// ---- Visualizations/Visualizations/Maintenance_2.TcVIS
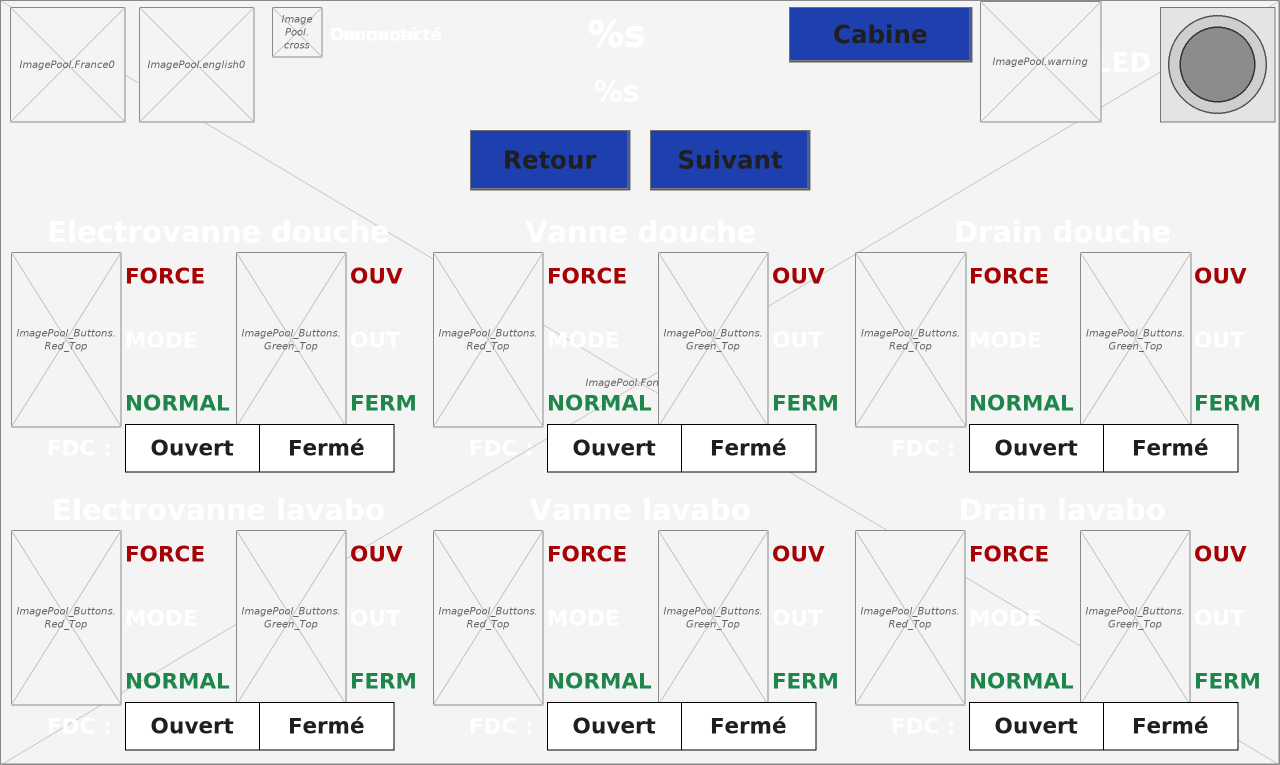
VISUALIZATION Maintenance_2  // 1280x765
    Frame (0,0 1280x765)
        shows masque()
    Button (650,130 160x60), "Suivant"
        OnMouseDown: execute {
            IF (Option_Bas_Debit OR Option_Douchette OR Option_NEP)
            	THEN
            	VisuElems.CURRENTVISU := 'Maintenance_3';
            	ELSIF (Option_WC_GV OR Option_WC_PV OR Option_Prise)
            		THEN
            		VisuElems.CURRENTVISU := 'Maintenance_4';
            	ELSIF (Option_Cabine_Climatique)
            		THEN
            		VisuElems.CURRENTVISU := 'Maintenance_5';
            	ELSIF (Option_Com_RegSouf_Ultrason)
            		THEN
            		VisuElems.CURRENTVISU := 'Maintenance_6';
            	ELSE
            		VisuElems.CURRENTVISU := 'Maintenance_7';
            END_IF
        }
    Button (470,130 160x60), "Retour"
        OnMouseDown: execute {
            IF (Option_RegSouf_Ultrason OR Option_Reg_Etanche_Ext OR Option_V3V_EauMitig)
            	THEN
            	VisuElems.CURRENTVISU := 'Maintenance_1';
            	ELSE
            	VisuElems.CURRENTVISU := 'menu';
            END_IF
        }
    Group (433,212 415x260), invisible if: NOT Option_Douche OR Option_Debitmetre_Douche
        Group (0,40 415x174)
            Group (0,0 225x175)
                Group (0,0 110x175)
                    Image (0,0 110x175), invisible if: EF_Cmd_Vanne_Alim_Douche, image: ImagePool_Buttons.Green_Bottom
                        OnMouseDown: toggle EF_Cmd_Vanne_Alim_Douche
                    Image (0,0 110x175), invisible if: NOT EF_Cmd_Vanne_Alim_Douche, image: ImagePool_Buttons.Red_Top
                        OnMouseDown: toggle EF_Cmd_Vanne_Alim_Douche
                Rectangle (111,0 114x48), "FORCE"
                Rectangle (111,64 114x48), "MODE"
                Rectangle (111,127 114x48), "NORMAL"
            Group (225,0 190x175), invisible if: NOT EF_Cmd_Vanne_Alim_Douche
                Group (0,0 110x175)
                    Image (0,0 110x175), invisible if: F_Cmd_Vanne_Alim_Douche, image: ImagePool_Buttons.Red_Bottom
                        OnMouseDown: toggle F_Cmd_Vanne_Alim_Douche
                    Image (0,0 110x175), invisible if: NOT F_Cmd_Vanne_Alim_Douche, image: ImagePool_Buttons.Green_Top
                        OnMouseDown: toggle F_Cmd_Vanne_Alim_Douche
                Rectangle (111,0 79x48), "OUV"
                Rectangle (111,64 79x48), "OUT"
                Rectangle (111,127 79x48), "FERM"
        Group (33,212 350x48)
            Rectangle (0,0 81x48), "FDC :"
            RoundedRectangle (81,0 135x48), "Ouvert", invisible if: NOT E_Vanne_Alim_Douche_Ouv
            RoundedRectangle (215,0 135x48), "Fermé", invisible if: NOT E_Vanne_Alim_Douche_Ferm
        Rectangle (0,0 415x40), "Vanne douche"
    Group (433,490 415x260), invisible if: NOT Option_Lavabo OR Option_Debitmetre_Lavabo
        Group (0,40 415x174)
            Group (0,0 225x175)
                Group (0,0 110x175)
                    Image (0,0 110x175), invisible if: EF_Cmd_Vanne_Alim_Douche, image: ImagePool_Buttons.Green_Bottom
                        OnMouseDown: toggle EF_Cmd_Vanne_Alim_Douche
                    Image (0,0 110x175), invisible if: NOT EF_Cmd_Vanne_Alim_Douche, image: ImagePool_Buttons.Red_Top
                        OnMouseDown: toggle EF_Cmd_Vanne_Alim_Douche
                Rectangle (111,0 114x48), "FORCE"
                Rectangle (111,64 114x48), "MODE"
                Rectangle (111,127 114x48), "NORMAL"
            Group (225,0 190x175), invisible if: NOT EF_Cmd_Vanne_Alim_Douche
                Group (0,0 110x175)
                    Image (0,0 110x175), invisible if: F_Cmd_Vanne_Alim_Douche, image: ImagePool_Buttons.Red_Bottom
                        OnMouseDown: toggle F_Cmd_Vanne_Alim_Douche
                    Image (0,0 110x175), invisible if: NOT F_Cmd_Vanne_Alim_Douche, image: ImagePool_Buttons.Green_Top
                        OnMouseDown: toggle F_Cmd_Vanne_Alim_Douche
                Rectangle (111,0 79x48), "OUV"
                Rectangle (111,64 79x48), "OUT"
                Rectangle (111,127 79x48), "FERM"
        Group (33,212 350x48)
            Rectangle (0,0 81x48), "FDC :"
            RoundedRectangle (81,0 135x48), "Ouvert", invisible if: NOT E_Vanne_Alim_Lavabo_Ouv
            RoundedRectangle (215,0 135x48), "Fermé", invisible if: NOT E_Vanne_Alim_Lavabo_Ferm
        Rectangle (0,0 415x40), "Vanne lavabo"
    Group (855,212 415x260), invisible if: NOT Option_Douche
        Group (0,40 415x174)
            Group (0,0 225x175)
                Group (0,0 110x175)
                    Image (0,0 111x175), invisible if: EF_Cmd_Vanne_Vid_Douche, image: ImagePool_Buttons.Green_Bottom
                        OnMouseDown: toggle EF_Cmd_Vanne_Vid_Douche
                    Image (0,0 111x175), invisible if: NOT EF_Cmd_Vanne_Vid_Douche, image: ImagePool_Buttons.Red_Top
                        OnMouseDown: toggle EF_Cmd_Vanne_Vid_Douche
                Rectangle (111,0 114x48), "FORCE"
                Rectangle (111,64 114x48), "MODE"
                Rectangle (111,127 114x48), "NORMAL"
            Group (225,0 190x175), invisible if: NOT EF_Cmd_Vanne_Vid_Douche
                Group (0,0 110x175)
                    Image (0,0 111x175), invisible if: F_Cmd_Vanne_Vid_Douche, image: ImagePool_Buttons.Red_Bottom
                        OnMouseDown: toggle F_Cmd_Vanne_Vid_Douche
                    Image (0,0 111x175), invisible if: NOT F_Cmd_Vanne_Vid_Douche, image: ImagePool_Buttons.Green_Top
                        OnMouseDown: toggle F_Cmd_Vanne_Vid_Douche
                Rectangle (111,0 79x48), "OUV"
                Rectangle (111,64 79x48), "OUT"
                Rectangle (111,127 79x48), "FERM"
        Group (33,212 350x48)
            Rectangle (0,0 81x48), "FDC :"
            RoundedRectangle (81,0 135x48), "Ouvert", invisible if: NOT E_Vanne_Vidange_Douche_Ouv
            RoundedRectangle (215,0 135x48), "Fermé", invisible if: NOT E_Vanne_Vidange_Douche_Ferm
        Rectangle (0,0 415x40), "Drain douche"
    Group (855,490 415x260), invisible if: NOT Option_Lavabo
        Group (0,40 415x174)
            Group (0,0 225x175)
                Group (0,0 110x175)
                    Image (0,0 110x175), invisible if: EF_Cmd_Vanne_Vid_Lavabo, image: ImagePool_Buttons.Green_Bottom
                        OnMouseDown: toggle EF_Cmd_Vanne_Vid_Lavabo
                    Image (0,0 110x175), invisible if: NOT EF_Cmd_Vanne_Vid_Lavabo, image: ImagePool_Buttons.Red_Top
                        OnMouseDown: toggle EF_Cmd_Vanne_Vid_Lavabo
                Rectangle (111,0 114x48), "FORCE"
                Rectangle (111,64 114x48), "MODE"
                Rectangle (111,127 114x48), "NORMAL"
            Group (225,0 190x175), invisible if: NOT EF_Cmd_Vanne_Vid_Lavabo
                Group (0,0 110x175)
                    Image (0,0 110x175), invisible if: F_Cmd_Vanne_Vid_Lavabo, image: ImagePool_Buttons.Red_Bottom
                        OnMouseDown: toggle F_Cmd_Vanne_Vid_Lavabo
                    Image (0,0 110x175), invisible if: NOT F_Cmd_Vanne_Vid_Lavabo, image: ImagePool_Buttons.Green_Top
                        OnMouseDown: toggle F_Cmd_Vanne_Vid_Lavabo
                Rectangle (111,0 79x48), "OUV"
                Rectangle (111,64 79x48), "OUT"
                Rectangle (111,127 79x48), "FERM"
        Group (33,212 350x48)
            Rectangle (0,0 81x48), "FDC :"
            RoundedRectangle (81,0 135x48), "Ouvert", invisible if: NOT E_Vanne_Vidange_Lavabo_Ouv
            RoundedRectangle (215,0 135x48), "Fermé", invisible if: NOT E_Vanne_Vidange_Lavabo_Ferm
        Rectangle (0,0 415x40), "Drain lavabo"
    Group (11,212 415x260), invisible if: NOT Option_Douche OR NOT Option_Debitmetre_Douche
        Group (0,40 415x174)
            Group (0,0 225x175)
                Group (0,0 110x175)
                    Image (0,0 110x175), invisible if: EF_Cmd_ElectroValve_Alim_Douche, image: ImagePool_Buttons.Green_Bottom
                    Image (0,0 110x175), invisible if: NOT EF_Cmd_ElectroValve_Alim_Douche, image: ImagePool_Buttons.Red_Top
                Rectangle (111,0 114x48), "FORCE"
                Rectangle (111,64 114x48), "MODE"
                Rectangle (111,127 114x48), "NORMAL"
            Group (225,0 190x175), invisible if: NOT EF_Cmd_ElectroValve_Alim_Douche
                Group (0,0 110x175)
                    Image (0,0 110x175), invisible if: F_Cmd_ElectroValve_Alim_Douche, image: ImagePool_Buttons.Red_Bottom
                        OnMouseDown: toggle F_Cmd_ElectroValve_Alim_Douche
                    Image (0,0 110x175), invisible if: NOT F_Cmd_ElectroValve_Alim_Douche, image: ImagePool_Buttons.Green_Top
                        OnMouseDown: toggle F_Cmd_ElectroValve_Alim_Douche
                Rectangle (111,0 79x48), "OUV"
                Rectangle (111,64 79x48), "OUT"
                Rectangle (111,127 79x48), "FERM"
        Group (33,212 350x48), invisible if: TRUE
            Rectangle (0,0 81x48), "FDC :"
            RoundedRectangle (81,0 135x48), "Ouvert"
            RoundedRectangle (215,0 135x48), "Fermé"
        Rectangle (0,0 415x40), "Electrovanne douche"
    Group (11,490 415x260), invisible if: NOT Option_Lavabo OR NOT Option_Debitmetre_Lavabo
        Group (0,40 415x174)
            Group (0,0 225x175)
                Group (0,0 110x175)
                    Image (0,0 110x175), invisible if: EF_Cmd_ElectroValve_Alim_Lavabo, image: ImagePool_Buttons.Green_Bottom
                        OnMouseDown: toggle EF_Cmd_ElectroValve_Alim_Lavabo
                    Image (0,0 110x175), invisible if: NOT EF_Cmd_ElectroValve_Alim_Lavabo, image: ImagePool_Buttons.Red_Top
                        OnMouseDown: toggle EF_Cmd_ElectroValve_Alim_Lavabo
                Rectangle (111,0 114x48), "FORCE"
                Rectangle (111,64 114x48), "MODE"
                Rectangle (111,127 114x48), "NORMAL"
            Group (225,0 190x175), invisible if: NOT EF_Cmd_ElectroValve_Alim_Lavabo
                Group (0,0 110x175)
                    Image (0,0 110x175), invisible if: F_Cmd_ElectroValve_Alim_Lavabo, image: ImagePool_Buttons.Red_Bottom
                        OnMouseDown: toggle F_Cmd_ElectroValve_Alim_Lavabo
                    Image (0,0 110x175), invisible if: NOT F_Cmd_ElectroValve_Alim_Lavabo, image: ImagePool_Buttons.Green_Top
                        OnMouseDown: toggle F_Cmd_ElectroValve_Alim_Lavabo
                Rectangle (111,0 79x48), "OUV"
                Rectangle (111,64 79x48), "OUT"
                Rectangle (111,127 79x48), "FERM"
        Group (33,212 350x48), invisible if: TRUE
            Rectangle (0,0 81x48), "FDC :"
            RoundedRectangle (81,0 135x48), "Ouvert"
            RoundedRectangle (215,0 135x48), "Fermé"
        Rectangle (0,0 415x40), "Electrovanne lavabo"
END_VISUALIZATION

// ---- Visualizations/Visualizations/Maintenance_3.TcVIS
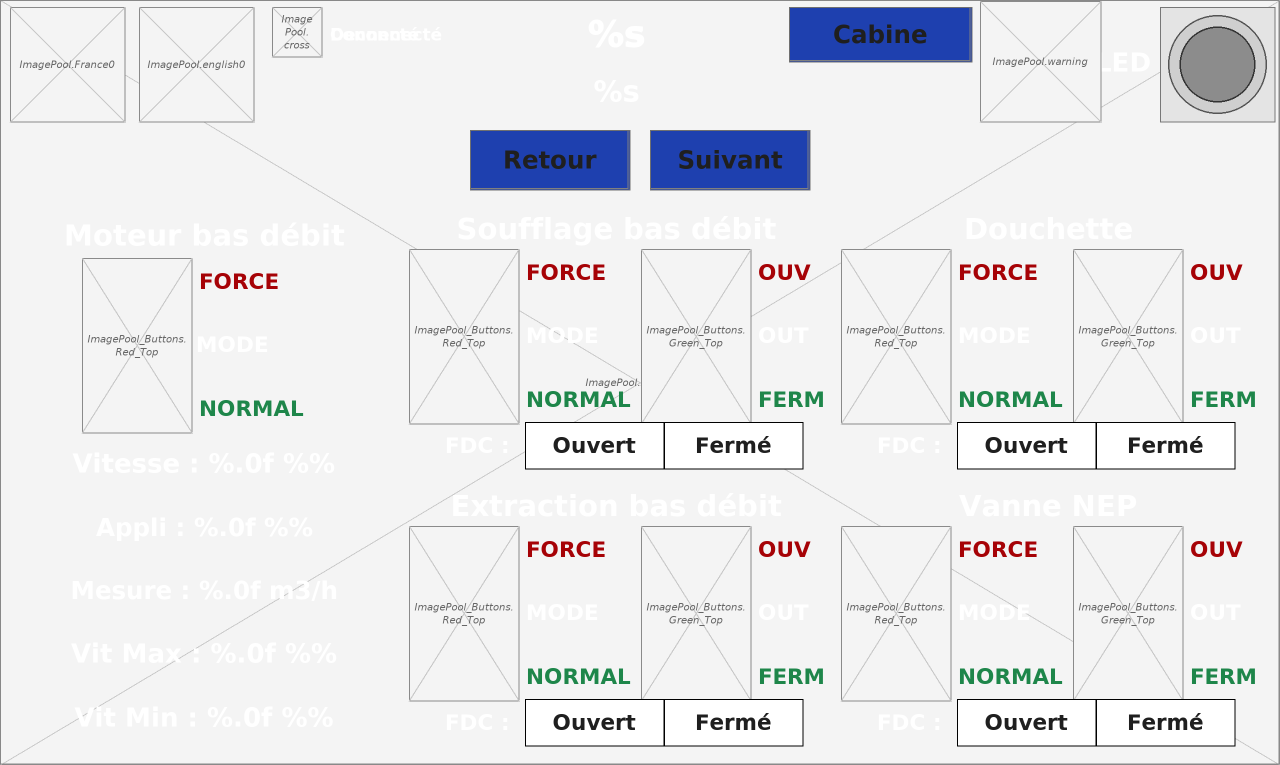
VISUALIZATION Maintenance_3  // 1280x765
    Frame (0,0 1280x765)
        shows masque()
    Group (409,209 415x260), invisible if: NOT Option_Bas_Debit
        Group (0,40 415x173)
            Group (0,0 232x174)
                Group (0,0 110x175)
                    Image (0,0 110x175), invisible if: EF_Vanne_Souf_Bas_Deb, image: ImagePool_Buttons.Green_Bottom
                        OnMouseDown: toggle EF_Vanne_Souf_Bas_Deb
                    Image (0,0 110x175), invisible if: NOT EF_Vanne_Souf_Bas_Deb, image: ImagePool_Buttons.Red_Top
                        OnMouseDown: toggle EF_Vanne_Souf_Bas_Deb
                Rectangle (114,0 118x47), "FORCE"
                Rectangle (114,63 118x47), "MODE"
                Rectangle (114,127 118x47), "NORMAL"
            Group (232,0 196x174), invisible if: NOT EF_Vanne_Souf_Bas_Deb
                Group (0,0 110x175)
                    Image (0,0 110x175), invisible if: F_Vanne_Souf_Bas_Deb, image: ImagePool_Buttons.Red_Bottom
                        OnMouseDown: toggle F_Vanne_Souf_Bas_Deb
                    Image (0,0 110x175), invisible if: NOT F_Vanne_Souf_Bas_Deb, image: ImagePool_Buttons.Green_Top
                        OnMouseDown: toggle F_Vanne_Souf_Bas_Deb
                Rectangle (114,0 82x47), "OUV"
                Rectangle (114,63 82x47), "OUT"
                Rectangle (114,127 82x47), "FERM"
        Group (33,213 350x47)
            Rectangle (0,0 83x47), "FDC :"
            RoundedRectangle (83,0 139x47), "Ouvert", invisible if: NOT E_Vanne_Souf_Bas_Deb_Ouv
            RoundedRectangle (222,0 139x47), "Fermé", invisible if: NOT E_Vanne_Souf_Bas_Deb_Ferm
        Rectangle (0,0 415x40), "Soufflage bas débit"
    Group (409,486 415x260), invisible if: NOT Option_Bas_Debit
        Group (0,40 415x173)
            Group (0,0 232x174)
                Group (0,0 110x175)
                    Image (0,0 110x175), invisible if: EF_Vanne_Ext_Bas_Deb, image: ImagePool_Buttons.Green_Bottom
                        OnMouseDown: toggle EF_Vanne_Ext_Bas_Deb
                    Image (0,0 110x175), invisible if: NOT EF_Vanne_Ext_Bas_Deb, image: ImagePool_Buttons.Red_Top
                        OnMouseDown: toggle EF_Vanne_Ext_Bas_Deb
                Rectangle (114,0 118x47), "FORCE"
                Rectangle (114,63 118x47), "MODE"
                Rectangle (114,127 118x47), "NORMAL"
            Group (232,0 196x174), text variable: NOT EF_Vanne_Ext_Bas_Deb, invisible if: NOT EF_Vanne_Ext_Bas_Deb
                Group (0,0 110x175)
                    Image (0,0 110x175), invisible if: F_Vanne_Ext_Bas_Deb, image: ImagePool_Buttons.Red_Bottom
                        OnMouseDown: toggle F_Vanne_Ext_Bas_Deb
                    Image (0,0 110x175), invisible if: NOT F_Vanne_Ext_Bas_Deb, image: ImagePool_Buttons.Green_Top
                        OnMouseDown: toggle F_Vanne_Ext_Bas_Deb
                Rectangle (114,0 82x47), "OUV"
                Rectangle (114,63 82x47), "OUT"
                Rectangle (114,127 82x47), "FERM"
        Group (33,213 350x47)
            Rectangle (0,0 83x47), "FDC :"
            RoundedRectangle (83,0 139x47), "Ouvert", invisible if: NOT E_Vanne_Ext_Bas_Deb_Ouv
            RoundedRectangle (222,0 139x47), "Fermé", invisible if: NOT E_Vanne_Ext_Bas_Deb_Ferm
        Rectangle (0,0 415x40), "Extraction bas débit"
    Group (841,209 415x260), invisible if: NOT Option_Douchette
        Group (0,40 415x173)
            Group (0,0 232x174)
                Group (0,0 110x175)
                    Image (0,0 110x175), invisible if: EF_Cmd_Vanne_Alim_Douchette, image: ImagePool_Buttons.Green_Bottom
                        OnMouseDown: toggle EF_Cmd_Vanne_Alim_Douchette
                    Image (0,0 110x175), invisible if: NOT EF_Cmd_Vanne_Alim_Douchette, image: ImagePool_Buttons.Red_Top
                        OnMouseDown: toggle EF_Cmd_Vanne_Alim_Douchette
                Rectangle (114,0 118x47), "FORCE"
                Rectangle (114,63 118x47), "MODE"
                Rectangle (114,127 118x47), "NORMAL"
            Group (232,0 196x174), invisible if: NOT EF_Cmd_Vanne_Alim_Douchette
                Group (0,0 110x175)
                    Image (0,0 110x175), invisible if: F_Cmd_Vanne_Alim_Douchette, image: ImagePool_Buttons.Red_Bottom
                        OnMouseDown: toggle F_Cmd_Vanne_Alim_Douchette
                    Image (0,0 110x175), invisible if: NOT F_Cmd_Vanne_Alim_Douchette, image: ImagePool_Buttons.Green_Top
                        OnMouseDown: toggle F_Cmd_Vanne_Alim_Douchette
                Rectangle (114,0 82x47), "OUV"
                Rectangle (114,63 82x47), "OUT"
                Rectangle (114,127 82x47), "FERM"
        Group (33,213 350x47)
            Rectangle (0,0 83x47), "FDC :"
            RoundedRectangle (83,0 139x47), "Ouvert", invisible if: NOT E_Vanne_Alim_Douchette_Ouv
            RoundedRectangle (222,0 139x47), "Fermé", invisible if: NOT E_Vanne_Alim_Douchette_Ferm
        Rectangle (0,0 415x40), "Douchette"
    Group (841,486 415x260), invisible if: NOT Option_NEP
        Group (0,40 415x173)
            Group (0,0 232x174)
                Group (0,0 110x175)
                    Image (0,0 110x175), invisible if: EF_Vanne_Alim_NEP, image: ImagePool_Buttons.Green_Bottom
                        OnMouseDown: toggle EF_Vanne_Alim_NEP
                    Image (0,0 110x175), invisible if: NOT EF_Vanne_Alim_NEP, image: ImagePool_Buttons.Red_Top
                        OnMouseDown: toggle EF_Vanne_Alim_NEP
                Rectangle (114,0 118x47), "FORCE"
                Rectangle (114,63 118x47), "MODE"
                Rectangle (114,127 118x47), "NORMAL"
            Group (232,0 196x174), invisible if: NOT EF_Vanne_Alim_NEP
                Group (0,0 110x175)
                    Image (0,0 110x175), invisible if: F_Vanne_Alim_NEP, image: ImagePool_Buttons.Red_Bottom
                        OnMouseDown: toggle F_Vanne_Alim_NEP
                    Image (0,0 110x175), invisible if: NOT F_Vanne_Alim_NEP, image: ImagePool_Buttons.Green_Top
                        OnMouseDown: toggle F_Vanne_Alim_NEP
                Rectangle (114,0 82x47), "OUV"
                Rectangle (114,63 82x47), "OUT"
                Rectangle (114,127 82x47), "FERM"
        Group (33,213 350x47)
            Rectangle (0,0 83x47), "FDC :"
            RoundedRectangle (83,0 139x47), "Ouvert", invisible if: NOT E_Vanne_Alim_NEP_Ouv
            RoundedRectangle (222,0 139x47), "Fermé", invisible if: NOT E_Vanne_Alim_NEP_Ferm
        Rectangle (0,0 415x40), "Vanne NEP"
    Button (650,130 160x60), "Suivant"
        OnMouseDown: execute {
            IF (Option_WC_GV OR Option_WC_PV OR Option_Prise)
            	THEN
            	VisuElems.CURRENTVISU := 'Maintenance_4';
            	ELSIF (Option_Cabine_Climatique)
            		THEN
            		VisuElems.CURRENTVISU := 'Maintenance_5';
            	ELSIF (Option_Com_RegSouf_Ultrason)
            		THEN
            		VisuElems.CURRENTVISU := 'Maintenance_6';
            	ELSE
            		VisuElems.CURRENTVISU := 'Maintenance_7';
            END_IF
        }
    Button (470,130 160x60), "Retour"
        OnMouseDown: execute {
            IF (Option_Douche OR Option_Lavabo)
            	THEN
            	VisuElems.CURRENTVISU := 'Maintenance_2';
            	ELSIF (Option_RegSouf_Ultrason OR Option_Reg_Etanche_Ext OR Option_V3V_EauMitig)
            		THEN
            		VisuElems.CURRENTVISU := 'Maintenance_1';
            	ELSE
            	VisuElems.CURRENTVISU := 'menu';
            END_IF
        }
    Group (15,204 380x545), invisible if: NOT Option_Bas_Debit
        Rectangle (0,0 379x63), "Moteur bas débit"
        Group (67,54 245x174)
            Group (0,0 110x175)
                Image (0,0 110x175), invisible if: Tab_Mot_Aerobox_Bas_Deb.Mot_Ecriture.0, image: ImagePool_Buttons.Green_Bottom
                    OnMouseDown: toggle Tab_Mot_Aerobox_Bas_Deb.Mot_Ecriture.0
                Image (0,0 110x175), invisible if: NOT Tab_Mot_Aerobox_Bas_Deb.Mot_Ecriture.0, image: ImagePool_Buttons.Red_Top
                    OnMouseDown: toggle Tab_Mot_Aerobox_Bas_Deb.Mot_Ecriture.0
            Rectangle (114,0 131x47), "FORCE"
            Rectangle (111,63 131x47), "MODE"
            Rectangle (114,127 131x47), "NORMAL"
        Rectangle (26,292 327x63), "Appli : %.0f %%", text variable: Cons_Actionneur_Moteur_BasDebit
        Rectangle (26,355 327x63), "Mesure : %.0f m3/h", text variable: MES_Petit_Debit_m3h_Extraction
        RoundedRectangle (2,228 374x63), "Vitesse : %.0f %%", text variable: Tab_Mot_Aerobox_Bas_Deb.W_ConsForcage, invisible if: NOT Tab_Mot_Aerobox_Bas_Deb.Mot_Ecriture.0
            OnMouseDown: write the text variable via VisuDialogs.Numpad, min 0, max 100, format %.0f
        RoundedRectangle (2,418 374x63), "Vit Max : %.0f %%", text variable: Tab_Mot_Aerobox_Bas_Deb.W_LimiteMaxCons
            OnMouseDown: write the text variable via VisuDialogs.Numpad, min 0, max 100, format %.0f
        RoundedRectangle (2,482 374x63), "Vit Min : %.0f %%", text variable: Tab_Mot_Aerobox_Bas_Deb.W_LimiteMinCons
            OnMouseDown: write the text variable via VisuDialogs.Numpad, min 0, max 100, format %.0f
END_VISUALIZATION

// ---- Visualizations/Visualizations/Maintenance_4.TcVIS
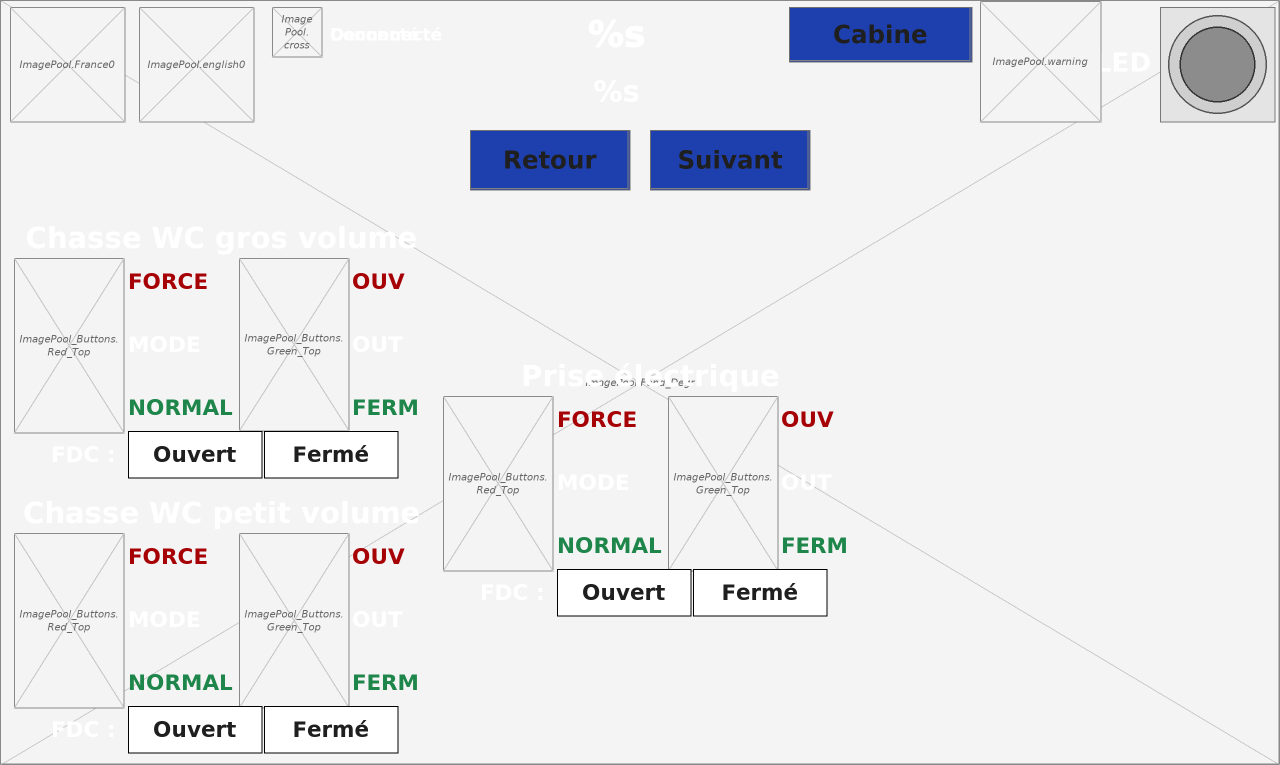
VISUALIZATION Maintenance_4  // 1280x765
    Frame (0,0 1280x765)
        shows masque()
    Button (470,130 160x60), "Retour"
        OnMouseDown: execute {
            IF (Option_Bas_Debit OR Option_Douchette OR Option_NEP)
            	THEN
            	VisuElems.CURRENTVISU := 'Maintenance_3';
            	ELSIF (Option_Douche OR Option_Lavabo)
            		THEN
            		VisuElems.CURRENTVISU := 'Maintenance_2';
            	ELSIF (Option_RegSouf_Ultrason OR Option_Reg_Etanche_Ext OR Option_V3V_EauMitig)
            		THEN
            		VisuElems.CURRENTVISU := 'Maintenance_1';
            	ELSE
            	VisuElems.CURRENTVISU := 'menu';
            END_IF
        }
    Button (650,130 160x60), "Suivant"
        OnMouseDown: execute {
            IF (Option_Cabine_Climatique)
            	THEN
            	VisuElems.CURRENTVISU := 'Maintenance_5';
            	ELSIF (Option_Com_RegSouf_Ultrason)
            		THEN
            		VisuElems.CURRENTVISU := 'Maintenance_6';
            	ELSE
            		VisuElems.CURRENTVISU := 'Maintenance_7';
            END_IF
        }
    Group (14,218 415x260), invisible if: NOT Option_WC_GV
        Group (0,40 415x173)
            Group (0,0 225x173)
                Group (0,0 110x175)
                    Image (0,0 110x175), text variable: EF_Cmd_Verin_WC_GV, invisible if: EF_Cmd_Verin_WC_GV, image: ImagePool_Buttons.Green_Bottom
                        OnMouseDown: toggle EF_Cmd_Verin_WC_GV
                    Image (0,0 110x175), text variable: NOT EF_Cmd_Verin_WC_GV, invisible if: NOT EF_Cmd_Verin_WC_GV, image: ImagePool_Buttons.Red_Top
                        OnMouseDown: toggle EF_Cmd_Verin_WC_GV
                Rectangle (111,0 114x47), "FORCE"
                Rectangle (111,63 114x47), "MODE"
                Rectangle (111,126 114x47), "NORMAL"
            Group (225,0 190x173), invisible if: NOT EF_Cmd_Verin_WC_GV
                Group (0,0 110x173)
                    Image (0,0 110x173), invisible if: F_Cmd_Verin_WC_GV, image: ImagePool_Buttons.Red_Bottom
                        OnMouseDown: toggle F_Cmd_Verin_WC_GV
                    Image (0,0 110x173), invisible if: NOT F_Cmd_Verin_WC_GV, image: ImagePool_Buttons.Green_Top
                        OnMouseDown: toggle F_Cmd_Verin_WC_GV
                Rectangle (110,0 80x47), "OUV"
                Rectangle (110,63 80x47), "OUT"
                Rectangle (110,126 80x47), "FERM"
        Group (34,213 350x47), invisible if: TRUE
            Rectangle (0,0 80x47), "FDC :"
            RoundedRectangle (80,0 134x47), "Ouvert"
            RoundedRectangle (216,0 134x47), "Fermé"
        Rectangle (0,0 415x40), "Chasse WC gros volume"
    Group (14,493 415x260), invisible if: NOT Option_WC_PV
        Group (0,40 415x173)
            Group (0,0 225x173)
                Group (0,0 110x175)
                    Image (0,0 110x175), invisible if: EF_Cmd_Verin_WC_PV, image: ImagePool_Buttons.Green_Bottom
                        OnMouseDown: toggle EF_Cmd_Verin_WC_PV
                    Image (0,0 110x175), invisible if: NOT EF_Cmd_Verin_WC_PV, image: ImagePool_Buttons.Red_Top
                        OnMouseDown: toggle EF_Cmd_Verin_WC_PV
                Rectangle (111,0 114x47), "FORCE"
                Rectangle (111,63 114x47), "MODE"
                Rectangle (111,126 114x47), "NORMAL"
            Group (225,0 190x173), invisible if: NOT EF_Cmd_Verin_WC_PV
                Group (0,0 110x175)
                    Image (0,0 110x175), invisible if: F_Cmd_Verin_WC_PV, image: ImagePool_Buttons.Red_Bottom
                        OnMouseDown: toggle F_Cmd_Verin_WC_PV
                    Image (0,0 110x175), invisible if: NOT F_Cmd_Verin_WC_PV, image: ImagePool_Buttons.Green_Top
                        OnMouseDown: toggle F_Cmd_Verin_WC_PV
                Rectangle (110,0 80x47), "OUV"
                Rectangle (110,63 80x47), "OUT"
                Rectangle (110,126 80x47), "FERM"
        Group (34,213 350x47), invisible if: TRUE
            Rectangle (0,0 80x47), "FDC :"
            RoundedRectangle (80,0 134x47), "Ouvert"
            RoundedRectangle (216,0 134x47), "Fermé"
        Rectangle (0,0 415x40), "Chasse WC petit volume"
    Group (443,356 415x260), invisible if: NOT Option_Prise
        Group (0,40 415x173)
            Group (0,0 225x173)
                Group (0,0 110x175)
                    Image (0,0 110x175), invisible if: EF_Cmd_PC_Cab, image: ImagePool_Buttons.Green_Bottom
                        OnMouseDown: toggle EF_Cmd_PC_Cab
                    Image (0,0 110x175), invisible if: NOT EF_Cmd_PC_Cab, image: ImagePool_Buttons.Red_Top
                        OnMouseDown: toggle EF_Cmd_PC_Cab
                Rectangle (111,0 114x47), "FORCE"
                Rectangle (111,63 114x47), "MODE"
                Rectangle (111,126 114x47), "NORMAL"
            Group (225,0 190x173), invisible if: NOT EF_Cmd_PC_Cab
                Group (0,0 110x175)
                    Image (0,0 110x175), invisible if: F_Cmd_PC_Cab, image: ImagePool_Buttons.Red_Bottom
                        OnMouseDown: toggle F_Cmd_PC_Cab
                    Image (0,0 110x175), invisible if: NOT F_Cmd_PC_Cab, image: ImagePool_Buttons.Green_Top
                        OnMouseDown: toggle F_Cmd_PC_Cab
                Rectangle (110,0 80x47), "OUV"
                Rectangle (110,63 80x47), "OUT"
                Rectangle (110,126 80x47), "FERM"
        Group (34,213 350x47), invisible if: TRUE
            Rectangle (0,0 80x47), "FDC :"
            RoundedRectangle (80,0 134x47), "Ouvert"
            RoundedRectangle (216,0 134x47), "Fermé"
        Rectangle (0,0 415x40), "Prise électrique"
END_VISUALIZATION

// ---- Visualizations/Visualizations/Maintenance_5.TcVIS
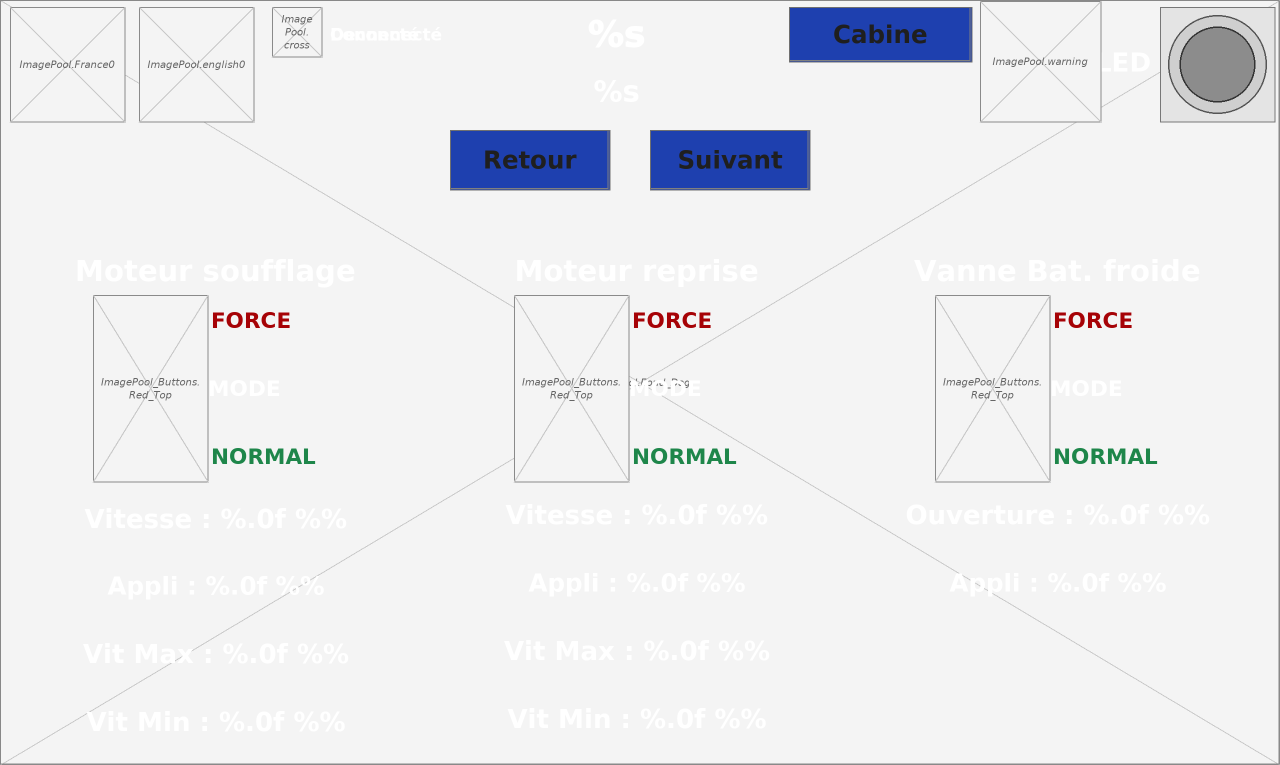
VISUALIZATION Maintenance_5  // 1280x765
    Frame (0,0 1280x765)
        shows masque()
    Button (450,130 160x60), "Retour"
        OnMouseDown: execute {
            IF (Option_WC_GV OR Option_WC_PV OR Option_Prise)
            	THEN
            	VisuElems.CURRENTVISU := 'Maintenance_4';
            	ELSIF (Option_Bas_Debit OR Option_Douchette OR Option_NEP)
            		THEN
            		VisuElems.CURRENTVISU := 'Maintenance_3';
            	ELSIF (Option_Douche OR Option_Lavabo)
            		THEN
            		VisuElems.CURRENTVISU := 'Maintenance_2';
            	ELSIF (Option_RegSouf_Ultrason OR Option_Reg_Etanche_Ext OR Option_V3V_EauMitig)
            		THEN
            		VisuElems.CURRENTVISU := 'Maintenance_1';
            	ELSE
            	VisuElems.CURRENTVISU := 'menu';
            END_IF
        }
    Button (650,130 160x60), "Suivant"
        OnMouseDown: execute {
            IF (Option_Com_RegSouf_Ultrason)
            	THEN
            		VisuElems.CURRENTVISU := 'Maintenance_6';
            	ELSE
            		VisuElems.CURRENTVISU := 'Maintenance_7';
            END_IF
        }
    Group (863,237 390x380), invisible if: NOT Option_Cabine_Climatique
        Rectangle (4,0 381x68), "Vanne Bat. froide"
        RoundedRectangle (0,244 390x68), "Ouverture : %.0f %%", text variable: F_Cons_V3V_Bat_Froid_CTA
            OnMouseDown: write the text variable via VisuDialogs.Numpad, min 0, max 100, format %.0f
        Rectangle (0,312 390x68), "Appli : %.0f %%", text variable: Cons_Actionneur_V3V_Froid_CTA
        Group (72,58 246x187)
            Group (0,0 115x187)
                Image (0,0 115x187), invisible if: EF_Cons_V3V_Bat_Froid_CTA, image: ImagePool_Buttons.Green_Bottom
                    OnMouseDown: toggle EF_Cons_V3V_Bat_Froid_CTA
                Image (0,0 115x187), invisible if: NOT EF_Cons_V3V_Bat_Froid_CTA, image: ImagePool_Buttons.Red_Top
                    OnMouseDown: toggle EF_Cons_V3V_Bat_Froid_CTA
            Rectangle (115,0 131x51), "FORCE"
            Rectangle (112,68 131x51), "MODE"
            Rectangle (115,136 131x51), "NORMAL"
    Group (21,237 390x519), invisible if: NOT Option_Cabine_Climatique
        Rectangle (4,0 381x68), "Moteur soufflage"
        RoundedRectangle (0,248 390x68), "Vitesse : %.0f %%", text variable: Tab_MotSouf_CTA.W_ConsForcage
            OnMouseDown: write the text variable via VisuDialogs.Numpad, min 0, max 100, format %.0f
        Rectangle (0,315 390x68), "Appli : %.0f %%", text variable: Tab_MotSouf_CTA.R_InfoCons
        Group (72,58 246x187)
            Group (0,0 115x187)
                Image (0,0 115x187), invisible if: Tab_MotSouf_CTA.Mot_Ecriture.0, image: ImagePool_Buttons.Green_Bottom
                    OnMouseDown: toggle Tab_MotSouf_CTA.Mot_Ecriture.0
                Image (0,0 115x187), invisible if: NOT Tab_MotSouf_CTA.Mot_Ecriture.0, image: ImagePool_Buttons.Red_Top
                    OnMouseDown: toggle Tab_MotSouf_CTA.Mot_Ecriture.0
            Rectangle (115,0 131x51), "FORCE"
            Rectangle (112,68 131x51), "MODE"
            Rectangle (115,136 131x51), "NORMAL"
        RoundedRectangle (0,383 390x68), "Vit Max : %.0f %%", text variable: Tab_MotSouf_CTA.W_LimiteMaxCons
            OnMouseDown: write the text variable via VisuDialogs.Numpad, min 0, max 100, format %.0f
        RoundedRectangle (0,451 390x68), "Vit Min : %.0f %%", text variable: Tab_MotSouf_CTA.W_LimiteMinCons
            OnMouseDown: write the text variable via VisuDialogs.Numpad, min 0, max 100, format %.0f
    Group (442,237 390x516), invisible if: NOT Option_Cabine_Climatique
        Rectangle (4,0 381x68), "Moteur reprise"
        RoundedRectangle (0,244 390x68), "Vitesse : %.0f %%", text variable: Tab_MotRep_CTA.W_ConsForcage
            OnMouseDown: write the text variable via VisuDialogs.Numpad, min 0, max 100, format %.0f
        Rectangle (0,312 390x68), "Appli : %.0f %%", text variable: Tab_MotRep_CTA.R_InfoCons
        Group (72,58 246x187)
            Group (0,0 115x187)
                Image (0,0 115x187), invisible if: Tab_MotRep_CTA.Mot_Ecriture.0, image: ImagePool_Buttons.Green_Bottom
                    OnMouseDown: toggle Tab_MotRep_CTA.Mot_Ecriture.0
                Image (0,0 115x187), invisible if: NOT Tab_MotRep_CTA.Mot_Ecriture.0, image: ImagePool_Buttons.Red_Top
                    OnMouseDown: toggle Tab_MotRep_CTA.Mot_Ecriture.0
            Rectangle (115,0 131x51), "FORCE"
            Rectangle (112,68 131x51), "MODE"
            Rectangle (115,136 131x51), "NORMAL"
        RoundedRectangle (0,448 390x68), "Vit Min : %.0f %%", text variable: Tab_MotRep_CTA.W_LimiteMinCons
            OnMouseDown: write the text variable via VisuDialogs.Numpad, min 0, max 100, format %.0f
        RoundedRectangle (0,380 390x68), "Vit Max : %.0f %%", text variable: Tab_MotRep_CTA.W_LimiteMaxCons
            OnMouseDown: write the text variable via VisuDialogs.Numpad, min 0, max 100, format %.0f
END_VISUALIZATION

// ---- Visualizations/Visualizations/Maintenance_6.TcVIS
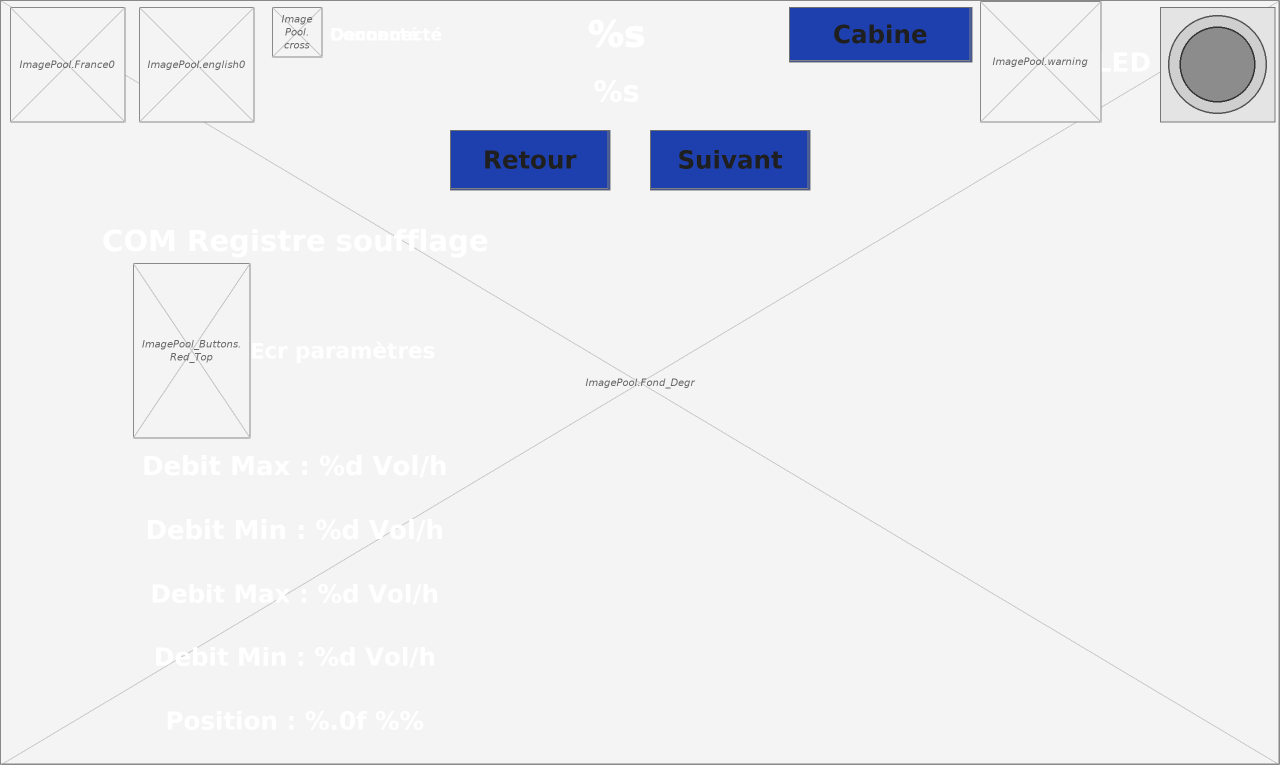
VISUALIZATION Maintenance_6  // 1280x765
    Frame (0,0 1280x765)
        shows masque()
    Button (650,130 160x60), "Suivant"
        OnMouseDown: change screen: Maintenance_7
    Button (450,130 160x60), "Retour"
        OnMouseDown: execute {
            IF (Option_Cabine_Climatique)
            	THEN
            	VisuElems.CURRENTVISU := 'Maintenance_5';
            	ELSIF (Option_WC_GV OR Option_WC_PV OR Option_Prise)
            		THEN
            		VisuElems.CURRENTVISU := 'Maintenance_4';
            	ELSIF (Option_Bas_Debit OR Option_Douchette OR Option_NEP)
            		THEN
            		VisuElems.CURRENTVISU := 'Maintenance_3';
            	ELSIF (Option_Douche OR Option_Lavabo)
            		THEN
            		VisuElems.CURRENTVISU := 'Maintenance_2';
            	ELSIF (Option_RegSouf_Ultrason OR Option_Reg_Etanche_Ext OR Option_V3V_EauMitig)
            		THEN
            		VisuElems.CURRENTVISU := 'Maintenance_1';
            	ELSE
            	VisuElems.CURRENTVISU := 'menu';
            END_IF
        }
    Group (64,209 463x544), invisible if: NOT Option_Com_RegSouf_Ultrason
        Rectangle (0,0 463x64), "COM Registre soufflage"
        Group (69,54 326x175)
            Group (0,0 117x175)
                Image (0,0 117x175), invisible if: Enable_ecr_param_Reg_Souf, image: ImagePool_Buttons.Green_Bottom
                    OnMouseDown: toggle Enable_ecr_param_Reg_Souf
                Image (0,0 117x175), invisible if: NOT Enable_ecr_param_Reg_Souf, image: ImagePool_Buttons.Red_Top
                    OnMouseDown: toggle Enable_ecr_param_Reg_Souf
            Rectangle (114,64 212x48), "Ecr paramètres"
        RoundedRectangle (32,225 398x64), "Debit Max : %d Vol/h", text variable: Ecriture_Cons_Max_Reg_Souf
            OnMouseDown: write the text variable via VisuDialogs.Numpad, min 0, max 1000, format %d
        Rectangle (32,353 398x64), "Debit Max : %d Vol/h", text variable: Lecture_Cons_Max_Reg_Souf
        Rectangle (32,416 398x64), "Debit Min : %d Vol/h", text variable: Lecture_Cons_Min_Reg_Souf
        RoundedRectangle (32,289 398x64), "Debit Min : %d Vol/h", text variable: Ecriture_Cons_Min_Reg_Souf
            OnMouseDown: write the text variable via VisuDialogs.Numpad, min 0, max 1000, format %d
        Rectangle (32,480 398x64), "Position : %.0f %%", text variable: MES_Pos_Reg_Souf
END_VISUALIZATION

// ---- Visualizations/Visualizations/Maintenance_7.TcVIS
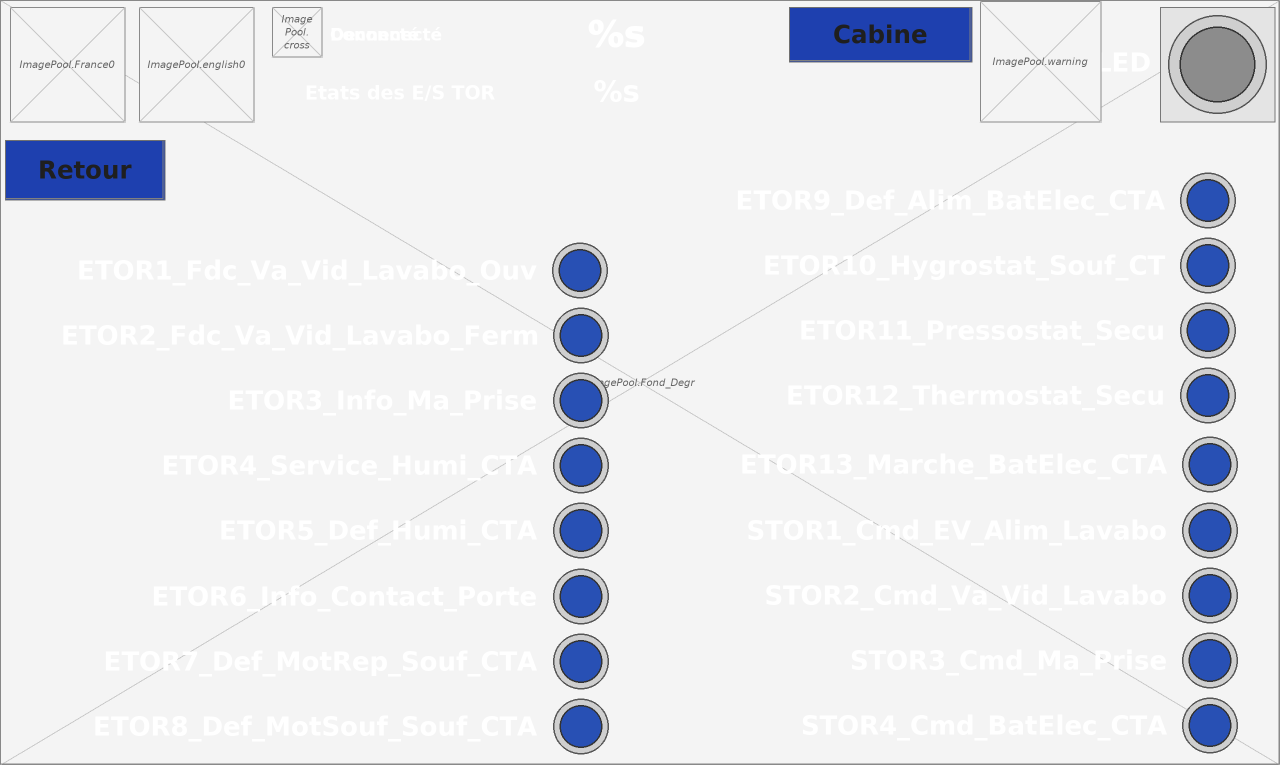
VISUALIZATION Maintenance_7  // 1280x765
    Frame (0,0 1280x765)
        shows masque()
    Rectangle (284,73 232x40), "Etats des E/S TOR"
    Button (5,140 160x60), "Retour", invisible if: Mode_Cabine_Depollution
        OnMouseDown: execute {
            IF (Option_Com_RegSouf_Ultrason)
            	THEN
            		VisuElems.CURRENTVISU := 'Maintenance_6';
            	ELSIF (Option_Cabine_Climatique)
            		THEN
            		VisuElems.CURRENTVISU := 'Maintenance_5';
            	ELSIF (Option_WC_GV OR Option_WC_PV OR Option_Prise)
            		THEN
            		VisuElems.CURRENTVISU := 'Maintenance_4';
            	ELSIF (Option_Bas_Debit OR Option_Douchette OR Option_NEP)
            		THEN
            		VisuElems.CURRENTVISU := 'Maintenance_3';
            	ELSIF (Option_Douche OR Option_Lavabo)
            		THEN
            		VisuElems.CURRENTVISU := 'Maintenance_2';
            	ELSIF (Option_RegSouf_Ultrason OR Option_Reg_Etanche_Ext OR Option_V3V_EauMitig)
            		THEN
            		VisuElems.CURRENTVISU := 'Maintenance_1';
            	ELSE
            	VisuElems.CURRENTVISU := 'menu';
            END_IF
        }
    Rectangle (7,238 533x65), "ETOR1_Fdc_Va_Vid_Lavabo_Ouv"
    Rectangle (9,303 533x65), "ETOR2_Fdc_Va_Vid_Lavabo_Ferm"
    Rectangle (7,368 533x65), "ETOR3_Info_Ma_Prise"
    Rectangle (7,433 533x65), "ETOR4_Service_Humi_CTA"
    Rectangle (7,498 533x65), "ETOR5_Def_Humi_CTA"
    Rectangle (7,564 533x65), "ETOR6_Info_Contact_Porte"
    Rectangle (7,629 533x65), "ETOR7_Def_MotRep_Souf_CTA"
    Rectangle (7,694 533x65), "ETOR8_Def_MotSouf_Souf_CTA"
    Rectangle (637,432 533x65), "ETOR13_Marche_BatElec_CTA"
    Rectangle (637,498 533x65), "STOR1_Cmd_EV_Alim_Lavabo"
    Rectangle (637,563 533x65), "STOR2_Cmd_Va_Vid_Lavabo"
    Rectangle (637,628 533x65), "STOR3_Cmd_Ma_Prise"
    Rectangle (637,693 533x65), "STOR4_Cmd_BatElec_CTA"
    Lamp1 (548,238 64x65), variable: ETOR1_Fdc_Va_Vid_Lavabo_Ouv, style: Lamp-Lamp1-Blue
    Lamp1 (549,303 64x65), variable: ETOR2_Fdc_Va_Vid_Lavabo_Ferm, style: Lamp-Lamp1-Blue
    Lamp1 (549,368 64x65), variable: ETOR3_Info_Ma_Prise, style: Lamp-Lamp1-Blue
    Lamp1 (549,433 64x65), variable: ETOR4_Service_Humi_CTA, style: Lamp-Lamp1-Blue
    Lamp1 (549,498 64x65), variable: ETOR5_Def_Humi_CTA, style: Lamp-Lamp1-Blue
    Lamp1 (549,564 64x65), variable: ETOR6_Info_Contact_Porte, style: Lamp-Lamp1-Blue
    Lamp1 (549,629 64x65), variable: ETOR7_Def_MotRep_Souf_CTA, style: Lamp-Lamp1-Blue
    Lamp1 (549,694 64x65), variable: ETOR8_Def_MotSouf_Souf_CTA, style: Lamp-Lamp1-Blue
    Lamp1 (1178,432 64x65), variable: ETOR13_Marche_BatElec_CTA, style: Lamp-Lamp1-Blue
    Lamp1 (1178,498 64x65), variable: STOR1_Cmd_EV_Alim_Lavabo, style: Lamp-Lamp1-Blue
    Lamp1 (1178,563 64x65), variable: STOR2_Cmd_Va_Vid_Lavabo, style: Lamp-Lamp1-Blue
    Lamp1 (1178,628 64x65), variable: STOR3_Cmd_Ma_Prise, style: Lamp-Lamp1-Blue
    Lamp1 (1178,693 64x65), variable: STOR4_Cmd_BatElec_CTA, style: Lamp-Lamp1-Blue
    Rectangle (635,168 533x65), "ETOR9_Def_Alim_BatElec_CTA"
    Lamp1 (1176,168 64x65), variable: ETOR9_Def_Alim_BatElec_CTA, style: Lamp-Lamp1-Blue
    Rectangle (635,233 533x65), "ETOR10_Hygrostat_Souf_CT"
    Lamp1 (1176,233 64x65), variable: ETOR10_Hygrostat_Souf_CT, style: Lamp-Lamp1-Blue
    Rectangle (635,298 533x65), "ETOR11_Pressostat_Secu"
    Lamp1 (1176,298 64x65), variable: ETOR11_Pressostat_Secu, style: Lamp-Lamp1-Blue
    Rectangle (635,363 533x65), "ETOR12_Thermostat_Secu"
    Lamp1 (1176,363 64x65), variable: ETOR12_Thermostat_Secu, style: Lamp-Lamp1-Blue
END_VISUALIZATION

// ---- Visualizations/Visualizations/Mes_Textes/Noms_Modes.TcTLO
TEXTLIST Noms_Modes
  1 = 'DOUCHE BONDE OUVERTE ET TEMPO' | En: 'SHOWER WITH DRAIN AND DELAY'
  2 = 'DOUCHE BONDE FERMEE ET TEMPO' | En: 'SHOWER WITHOUT DRAIN AND DELAY'
  3 = 'DOUCHETTE' | En: 'CLEANING'
  4 = 'LAVABO BONDE OUVERTE ET TEMPO' | En: 'SINK WITH DRAIN AND DELAY'
  5 = 'LAVABO BONDE FERMEE ET TEMPO' | En: 'SINK WITHOUT DRAIN AND DELAY'
  6 = 'PRISE ELECTRIQUE' | En: 'PLUG ACTIVATE'
  7 = 'VIDANGE(S)' | En: 'OPENED DRAIN'
  8 = 'NEUTRE' | En: 'NEUTRAL'
  9 = 'CHASSE D EAU GRAND VOLUME' | En: 'LARGE VOLUME TOILET FLUSH'
  10 = 'DEPOLLUTION' | En: 'DECONTAMINATION'
  11 = 'NEUTRE AVEC BAS DEBIT' | En: 'NEUTRAL WITH LOW FLOW'
  12 = 'DOUCHE BONDE OUVERTE ET VOLUME' | En: 'SHOWER WITH DRAIN AND VOLUME'
  13 = 'DOUCHE BONDE FERMEE ET VOLUME' | En: 'SHOWER WITHOUT DRAIN AND VOLUME'
  14 = 'LAVABO BONDE OUVERTE ET VOLUME' | En: 'SINK WITH DRAIN AND VOLUME'
  15 = 'LAVABO BONDE FERMEE ET VOLUME' | En: 'SINK WITHOUT DRAIN AND VOLUME'
  16 = 'DOUCHE BONDE OUVERTE ET BOUTON' | En: 'SHOWER WITH DRAIN AND BUTTON'
  17 = 'LAVABO BONDE OUVERTE ET BOUTON' | En: 'SINK WITH DRAIN AND BUTTON'
  18 = 'LAVAGE CHAUD' | En: 'HOT CLEANING'
  19 = 'LAVAGE FROID' | En: 'COLD CLEANING'
  20 = 'MODE PARAMETRABLE' | En: 'PARAMETER MODE'
  21 = 'ALERTE PREPARATEUR' | En: 'PREPARATOR ALERT'
  22 = 'ALERTE EVALUATEUR' | En: 'EVALUATOR ALERT'
  23 = 'EVALUATION' | En: 'EVALUATION'
  24 = 'EVALUATION AVEC AIR' | En: 'EVALUATION WITH AIR FLOW'
  25 = 'MISE EN CONDITION' | En: 'CONDITIONING BOOTH'
  26 = 'CHASSE D EAU PETIT VOLUME' | En: 'SMALL VOLUME TOILET FLUSH'
  27 = 'LAVAGE NEP' | En: 'CLEANING'
  28 = 'CABINE EN CONDITION' | En: 'BOOTH IN CONDITION'
  29 = 'LIBRE' | En: 'EMPTY'
  30 = 'MODE TEXTE' | En: 'TEXT MODE'
  0 = ''
   = ''
END_TEXTLIST

// ---- Visualizations/Visualizations/ModeManuel.TcVIS
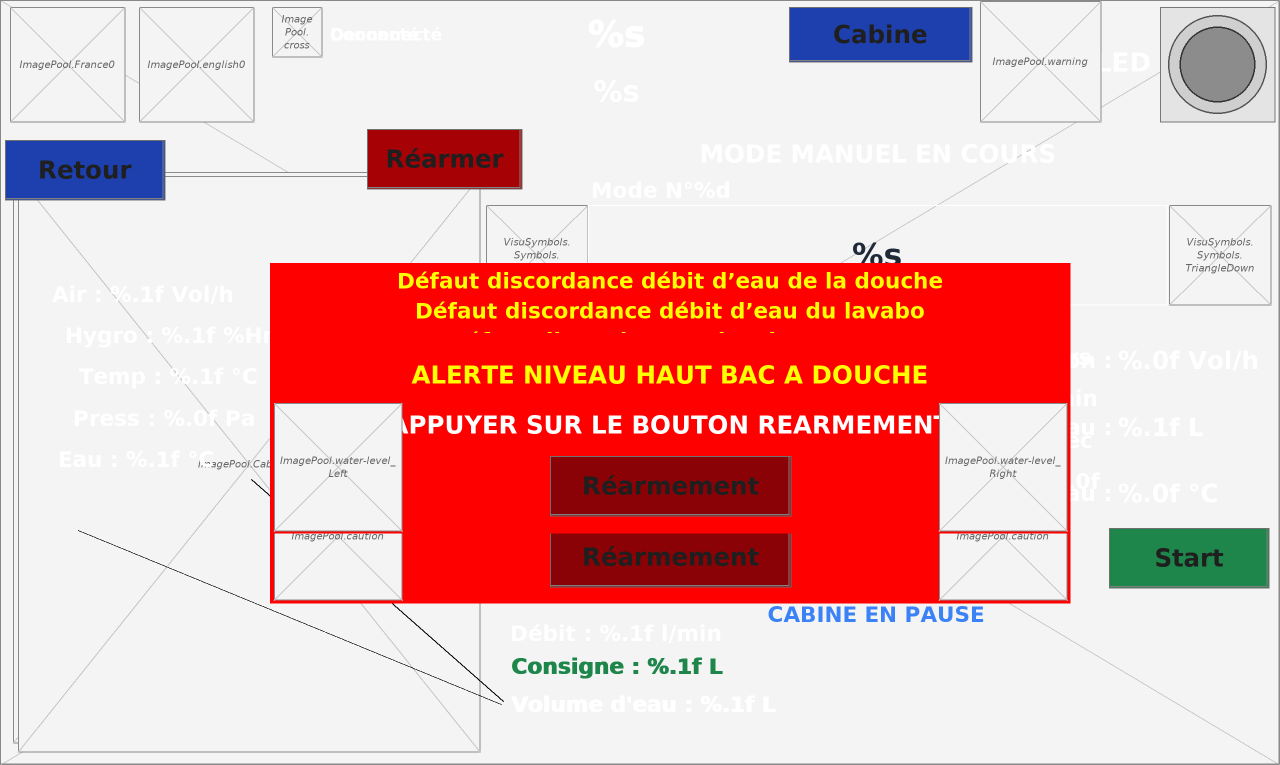
VISUALIZATION ModeManuel  // 1280x765
    Frame (0,0 1280x765)
        shows masque()
    Image (13,172 466x571), image: ImagePool.Cabine-2
    Polygon (40,654) (180,695) (321,730) (395,695) (469,654), colour variable: GVL_Visu.Couleur_Cabine
    Polygon (42,654) (40,249) (323,189) (466,256) (467,654), colour variable: GVL_Visu.Couleur_Cabine
    Image (18,176 462x576), image: ImagePool.Cabine_1
        OnMouseDown: OpenDialog Dialog=Actionneurs, OpenModal=True, OpenCentered=True
    Button (5,140 160x60), "Retour", invisible if: Mode_Cabine_Manuel
        OnMouseDown: change screen: menu
    Group (49,274 322x206)
        Rectangle (13,41 295x41), "Hygro : %.1f %Hr", text variable: Tab_MES_Sonde_Hygro_Amb.R_MesCor
        Rectangle (27,82 295x41), "Temp : %.1f °C", text variable: Tab_MES_Sonde_Temp_Amb.R_MesCor
        Rectangle (0,0 295x41), "Air : %.1f Vol/h", text variable: MES_Debit_Volh_Soufflage, invisible if: TRUE
        Rectangle (21,124 295x41), "Press : %.0f Pa", text variable: Tab_MES_Sonde_Press_Cab.R_MesCor
        Rectangle (6,165 295x41), "Eau : %.1f °C", text variable: MES_Temp_Eau_Mitige_General
    Rectangle (507,613 294x41), "Débit : %.1f l/min", text variable: GVL_Visu.Visu_Mes_Debit_Eau_Manu, invisible if: NOT GVL_Visu.Visu_Debit_Eau_Manu
    Group (486,205 100x100), invisible if: Mode_Cabine_Manuel
        OnMouseDown: execute {
            Manu_Choix_Numero_Mode := Manu_Choix_Numero_Mode - 1;
            IF (Manu_Choix_Numero_Mode < GVL_Visu.Min_Mode_Manu)
            	THEN
            	Manu_Choix_Numero_Mode := GVL_Visu.Min_Mode_Manu;
            END_IF
            GVL_Visu.Manu_i := 30;
            FOR GVL_Visu.Manu_i := 30 TO 0 BY -1 DO
            	IF ((NOT GVL_Visu.Tab_Choix_Modes[GVL_Visu.Manu_i]) AND (Manu_Choix_Numero_Mode = GVL_Visu.Manu_i))
            		THEN
            		Manu_Choix_Numero_Mode := Manu_Choix_Numero_Mode - 1;
            	END_IF
            END_FOR
        }
        Button (0,0 100x100)
        Image (0,0 102x100), image: VisuSymbols.Symbols.TriangleUp
    RoundedRectangle (588,205 579x100), "%s", text list: 'Noms_Modes', text index: GVL_Visu.Manu_Choix_Numero_Mode_INT
    Group (1169,205 100x100), invisible if: Mode_Cabine_Manuel
        OnMouseDown: execute {
            Manu_Choix_Numero_Mode := Manu_Choix_Numero_Mode + 1;
            GVL_Visu.Manu_j := 0;
            FOR GVL_Visu.Manu_j := 0 TO 29 BY 1 DO
            	IF (NOT (GVL_Visu.Tab_Choix_Modes[GVL_Visu.Manu_j]) AND (Manu_Choix_Numero_Mode = GVL_Visu.Manu_j))
            		THEN
            		Manu_Choix_Numero_Mode := Manu_Choix_Numero_Mode + 1;
            	END_IF
            END_FOR
            IF (Manu_Choix_Numero_Mode > GVL_Visu.Max_Mode_Manu)
            	THEN
            	Manu_Choix_Numero_Mode := GVL_Visu.Max_Mode_Manu;
            END_IF
        }
        Button (0,0 100x100)
        Image (0,0 102x100), image: VisuSymbols.Symbols.TriangleDown
    Button (367,129 155x60), "Réarmer", invisible if: NOT Condi_Affich_Rearm
        OnMouseDown: toggle Cmd_Rearmement
    Rectangle (588,170 186x41), "Mode N°%d", text variable: GVL_Visu.Manu_Choix_Numero_Mode_INT
    Button (1109,528 160x60), "Start", invisible if: Mode_Cabine_Manuel
        OnMouseDown: toggle Start_Mode_Manu
    Group (483,329 786x263), invisible if: Mode_Cabine_Manuel
        Group (445,67 341x63), invisible if: NOT GVL_Visu.Affich_Debit_Eau_Manu_Douche
            Rectangle (0,0 187x63), "Vol. d'eau :"
            RoundedRectangle (187,0 154x63), "%.1f L", text variable: Manu_Lct_Cons_Vol_Douche
                OnMouseDown: write the text variable via VisuDialogs.Numpad, min 0, max 100, format %0.1f
        Group (0,0 445x63), invisible if: GVL_Visu.Affich_Debit_Eau_Manu
            Rectangle (0,0 186x63), "Heure(s) :"
            RoundedRectangle (186,0 259x63), "%.0f heure(s)", text variable: Manu_Tempo_Transition_Heure
                OnMouseDown: write the text variable via VisuDialogs.Numpad, min 0, max 23, format %.0f
        Group (0,67 445x63), invisible if: GVL_Visu.Affich_Debit_Eau_Manu
            Rectangle (0,0 186x63), "Minute(s) :"
            RoundedRectangle (186,0 259x63), "%.0f minute(s)", text variable: Manu_Tempo_Transition_Minute
                OnMouseDown: write the text variable via VisuDialogs.Numpad, min 0, max 59, format %.0f
        Group (0,133 445x63), invisible if: GVL_Visu.Affich_Debit_Eau_Manu
            Rectangle (0,0 186x63), "Seconde(s) :"
            RoundedRectangle (186,0 259x63), "%.0f seconde(s)", text variable: Manu_Tempo_Transition_Seconde
                OnMouseDown: write the text variable via VisuDialogs.Numpad, min 0, max 59, format %.0f
        Group (445,0 341x63), invisible if: GVL_Visu.Manu_Choix_Numero_Mode_INT = 8
            Rectangle (0,0 187x63), "Ventilation :"
            RoundedRectangle (187,0 154x63), "%.0f Vol/h", text variable: Manu_Cons_Deb_Soufflage
                OnMouseDown: write the text variable via VisuDialogs.Numpad, min 0, max 200, format %.0f
        Group (0,200 445x63), invisible if: NOT GVL_Visu.Affich_ChasseEau_Manu
            Rectangle (0,0 186x63), "Nbre chasse :"
            RoundedRectangle (186,0 259x63), "%.0f", text variable: Manu_Cons_Nbre_Chasse
                OnMouseDown: write the text variable via VisuDialogs.Numpad, min 0, max 99, format %.0f
        Group (445,133 341x63), invisible if: NOT GVL_Visu.Visu_Temp_Manu
            Rectangle (0,0 187x63), "Temp. eau :"
            RoundedRectangle (187,0 154x63), "%.0f °C", text variable: Manu_Cons_Temp_Eau
                OnMouseDown: write the text variable via VisuDialogs.Numpad, min 10, max 50, format %.0f
        Group (445,67 341x63), invisible if: NOT GVL_Visu.Affich_Debit_Eau_Manu_Lavabo
            Rectangle (0,0 187x63), "Vol. d'eau :"
            RoundedRectangle (187,0 154x63), "%.1f L", text variable: Manu_Lct_Cons_Vol_Lavabo
                OnMouseDown: write the text variable via VisuDialogs.Numpad, min 0, max 100, format %0.1f
    Group (483,129 650x506), invisible if: NOT Mode_Cabine_Manuel
        Button (312,400 160x60), "Pause", invisible if: Statut_Pause_Force
            OnMouseDown: toggle Bp_Pause
        Rectangle (140,0 510x50), "MODE MANUEL EN COURS", invisible if: GVL_Visu.On_Off_Anim
        Button (0,401 160x60), "Stop"
            OnMouseDown: toggle Reset_Mode_Manu
        Button (312,400 160x60), "Re-Start", invisible if: NOT Statut_Pause_Force
            OnMouseDown: toggle Bp_Pause
        Group (172,208 446x165), invisible if: GVL_Visu.Affich_Debit_Eau_Manu
            Rectangle (11,0 322x41), "Heure(s) restante(s) :"
            Rectangle (333,0 113x41), "%.0f hrs", text variable: Temp_Restant_Heure
            Rectangle (11,83 322x41), "Seconde(s) restante(s) :"
            Rectangle (333,83 113x41), "%.0f sec", text variable: Temp_Restant_Seconde
            Rectangle (11,41 322x41), "Minute(s) restante(s) :"
            Rectangle (333,41 113x41), "%.0f min", text variable: Temp_Restant_Minute
            Group (0,124 446x41), invisible if: NOT GVL_Visu.Visu_ChasseEau_Manu
                Rectangle (0,0 322x41), "Chasse(s) restante(s) :"
                Rectangle (322,0 74x41), "%.0f /", text variable: Nbre_Chasse_EnCours
                Rectangle (388,0 58x41), "%.0f", text variable: Nbre_Chasse_Total
        Rectangle (246,465 294x41), "CABINE EN PAUSE", invisible if: GVL_Visu.On_Off_Anim OR NOT Comande_Pause
    Group (251,479 602x246), invisible if: NOT GVL_Visu.Visu_VolEau_Douche_Manu
        Line (0,0) (252,222)
        Rectangle (258,205 344x41), "Volume d'eau : %.1f L", text variable: Lect_Volume_Eau_Douche
        Rectangle (258,171 344x33), "Consigne : %.1f L", text variable: Manu_Lct_Cons_Vol_Douche
    Group (78,530 774x195), invisible if: NOT GVL_Visu.Visu_VolEau_Lavabo_Manu
        Line (0,0) (423,174)
        Rectangle (430,154 344x41), "Volume d'eau : %.1f L", text variable: Lect_Volume_Eau_Lavabo
        Rectangle (430,120 344x33), "Consigne : %.1f L", text variable: Manu_Lct_Cons_Vol_Lavabo
    Group (270,263 800x340)
        Frame (0,0 800x340), invisible if: NOT GVL_Visu.Affichage_PopUp_Alarm
            shows PopUp_Alarms()
        Frame (0,70 800x200), invisible if: NOT GVL_Visu.Affichage_PopUp_HightLevel
            shows PopUp_Hight_Level()
END_VISUALIZATION

// ---- Visualizations/Visualizations/Nettoyage.TcVIS
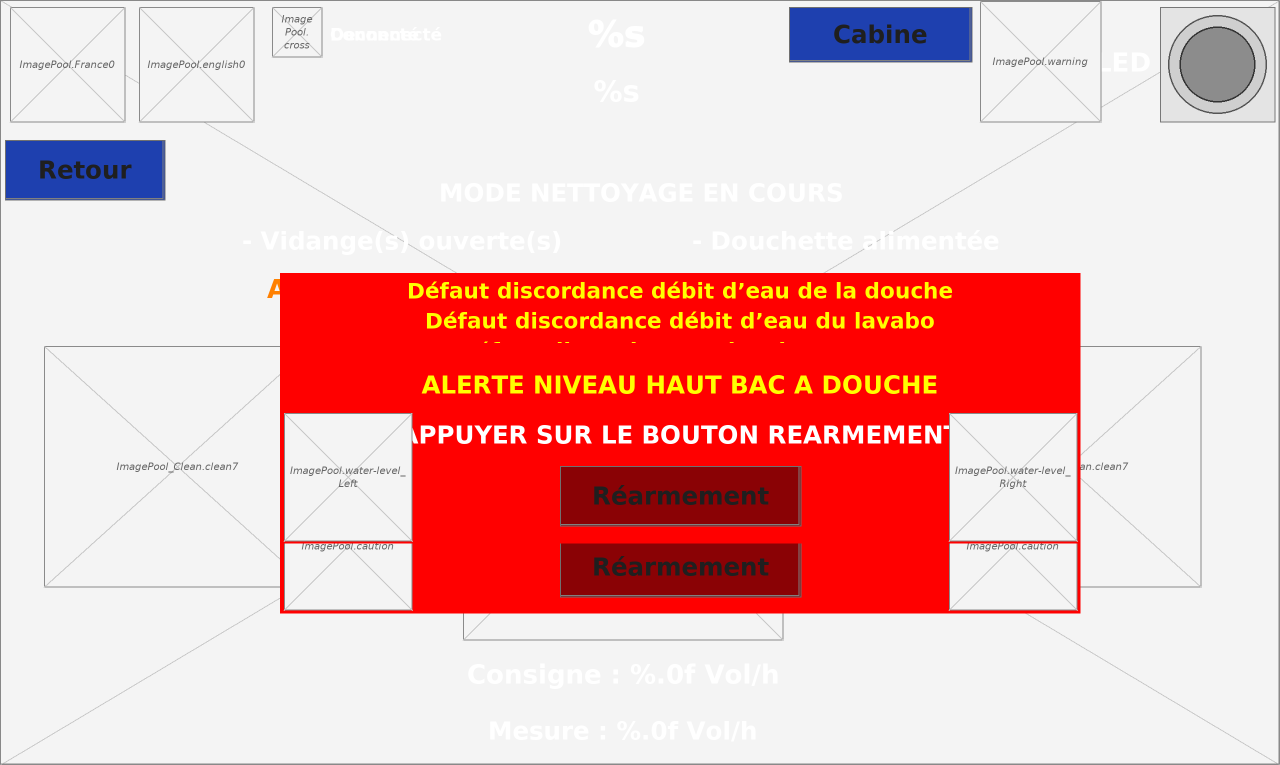
VISUALIZATION Nettoyage  // 1280x765
    Frame (0,0 1280x765)
        shows masque()
    Rectangle (384,706 478x50), "Mesure : %.0f Vol/h", text variable: MES_Debit_Volh_Soufflage
    Group (44,346 267x241)
        Image (0,0 267x241), text variable: NOT GVL_Visu.Cmd_Img_Clean1, invisible if: NOT GVL_Visu.Cmd_Img_Clean1, image: ImagePool_Clean.clean1
        Image (0,0 267x241), text variable: NOT GVL_Visu.Cmd_Img_Clean2, invisible if: NOT GVL_Visu.Cmd_Img_Clean2, image: ImagePool_Clean.clean2
        Image (0,0 267x241), text variable: NOT GVL_Visu.Cmd_Img_Clean3, invisible if: NOT GVL_Visu.Cmd_Img_Clean3, image: ImagePool_Clean.clean3
        Image (0,0 267x241), text variable: NOT GVL_Visu.Cmd_Img_Clean4, invisible if: NOT GVL_Visu.Cmd_Img_Clean4, image: ImagePool_Clean.clean4
        Image (0,0 267x241), text variable: NOT GVL_Visu.Cmd_Img_Clean4, invisible if: NOT GVL_Visu.Cmd_Img_Clean5, image: ImagePool_Clean.clean5
        Image (0,0 267x241), text variable: NOT GVL_Visu.Cmd_Img_Clean6, invisible if: NOT GVL_Visu.Cmd_Img_Clean6, image: ImagePool_Clean.clean6
        Image (0,0 267x241), text variable: NOT GVL_Visu.Cmd_Img_Clean7, invisible if: NOT GVL_Visu.Cmd_Img_Clean7, image: ImagePool_Clean.clean7
    Image (463,320 320x320), invisible if: NOT Start_Etat_Nettoyage, image: ImagePool_Buttons.Selecteur_left
        OnMouseDown: toggle Start_Etat_Nettoyage
    Image (463,320 320x320), invisible if: Start_Etat_Nettoyage, image: ImagePool_Buttons.Selecteur_right - Copie
        OnMouseDown: toggle Start_Etat_Nettoyage
    Rectangle (358,338 170x50), "Start"
    Rectangle (711,338 170x50), "Stop"
    Group (934,346 267x241)
        Image (0,0 267x241), text variable: NOT GVL_Visu.Cmd_Img_Clean1, invisible if: NOT GVL_Visu.Cmd_Img_Clean1, image: ImagePool_Clean.clean1
        Image (0,0 267x241), text variable: NOT GVL_Visu.Cmd_Img_Clean2, invisible if: NOT GVL_Visu.Cmd_Img_Clean2, image: ImagePool_Clean.clean2
        Image (0,0 267x241), text variable: NOT GVL_Visu.Cmd_Img_Clean3, invisible if: NOT GVL_Visu.Cmd_Img_Clean3, image: ImagePool_Clean.clean3
        Image (0,0 267x241), text variable: NOT GVL_Visu.Cmd_Img_Clean4, invisible if: NOT GVL_Visu.Cmd_Img_Clean4, image: ImagePool_Clean.clean4
        Image (0,0 267x241), text variable: NOT GVL_Visu.Cmd_Img_Clean4, invisible if: NOT GVL_Visu.Cmd_Img_Clean5, image: ImagePool_Clean.clean5
        Image (0,0 267x241), text variable: NOT GVL_Visu.Cmd_Img_Clean6, invisible if: NOT GVL_Visu.Cmd_Img_Clean6, image: ImagePool_Clean.clean6
        Image (0,0 267x241), text variable: NOT GVL_Visu.Cmd_Img_Clean7, invisible if: NOT GVL_Visu.Cmd_Img_Clean7, image: ImagePool_Clean.clean7
    Group (139,169 968x144), invisible if: NOT Mode_Cabine_Nettoyage
        Rectangle (160,0 685x48), "MODE NETTOYAGE EN COURS", invisible if: GVL_Visu.On_Off_Anim
        Rectangle (25,48 476x48), "- Vidange(s) ouverte(s)", invisible if: NOT E_Vanne_Vidange_Douche_Ouv
        Rectangle (469,48 476x48), "- Douchette alimentée", invisible if: NOT S_Cmd_Vanne_Alim_Douchette
        Rectangle (0,96 968x48), "APPUYER SUR LA DOUCHETTE POUR L'UTILISER !", invisible if: NOT S_Cmd_Vanne_Alim_Douchette
    RoundedRectangle (412,642 423x65), "Consigne : %.0f Vol/h", text variable: Cons_Deb_Souf_Etat_Nettoyage
        OnMouseDown: write the text variable via VisuDialogs.Numpad, min 0, max 23, format %.0f
    Button (5,140 160x60), "Retour", invisible if: Mode_Cabine_Nettoyage
        OnMouseDown: change screen: menu
    Group (280,273 800x340)
        Frame (0,0 800x340), invisible if: NOT GVL_Visu.Affichage_PopUp_Alarm
            shows PopUp_Alarms()
        Frame (0,70 800x200), invisible if: NOT GVL_Visu.Affichage_PopUp_HightLevel
            shows PopUp_Hight_Level()
END_VISUALIZATION

// ---- Visualizations/Visualizations/Maintenance_1.TcVIS
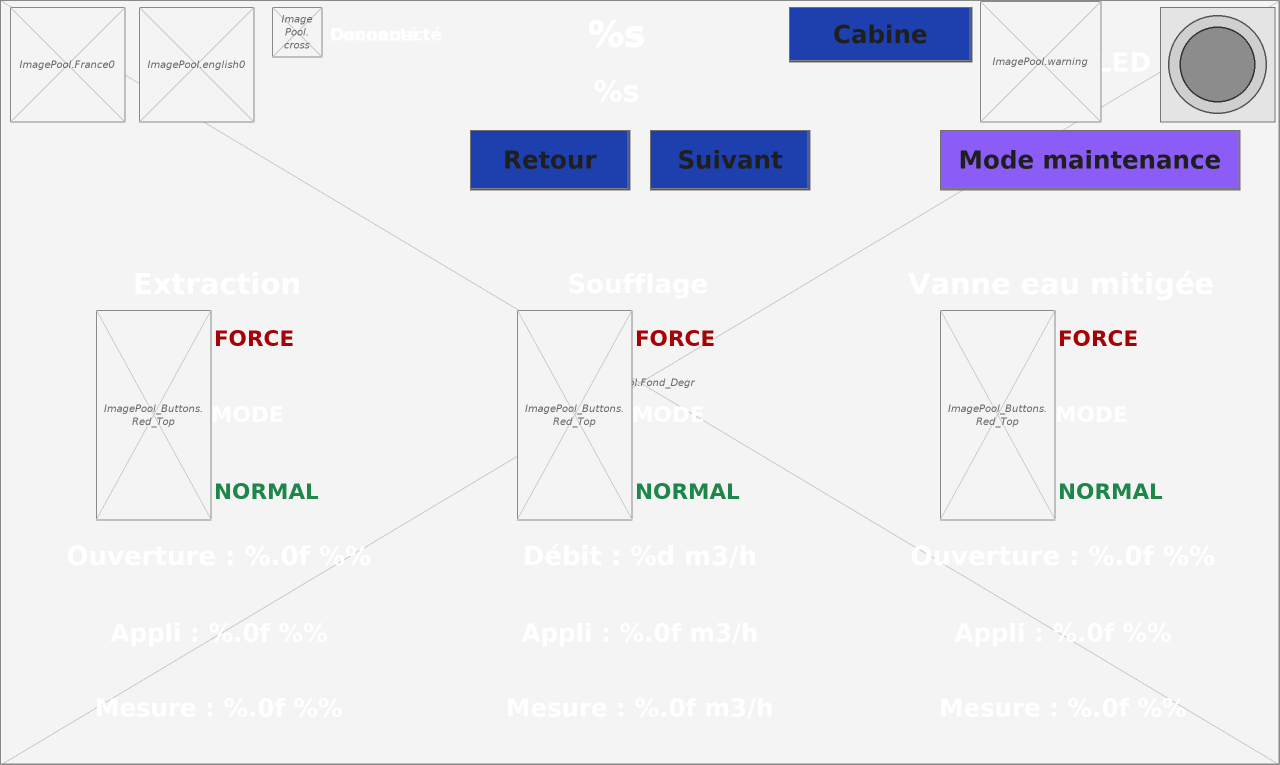
VISUALIZATION Maintenance_1  // 1280x765
    Frame (0,0 1280x765)
        shows masque()
    Button (470,130 160x60), "Retour"
        OnMouseDown: change screen: menu
        OnMouseDown: VisuUserMgmt Type=Logout
    Button (940,130 300x60), "Mode maintenance"
        OnMouseDown: toggle Cmd_Mode_Maintenance
    Group (445,246 390x500), invisible if: NOT Option_RegSouf_Ultrason
        Rectangle (3,0 380x76), "Soufflage"
        RoundedRectangle (0,272 390x76), "Débit : %d m3/h", text variable: F_Cons_Registre_Soufflage, invisible if: NOT EF_Cons_Registre_Soufflage
            OnMouseDown: write the text variable via VisuDialogs.Numpad, min 0, max 1000, format %d
        Rectangle (0,349 390x76), "Appli : %.0f m3/h", text variable: Cons_Actio_Registre_Souf_m3h
        Rectangle (0,424 390x76), "Mesure : %.0f m3/h", text variable: Tab_MES_Sonde_Gros_Debit_Soufflage.R_MesCor
        Group (72,64 246x208)
            Group (0,0 115x210)
                Image (0,0 115x210), invisible if: EF_Cons_Registre_Soufflage, image: ImagePool_Buttons.Green_Bottom
                    OnMouseDown: toggle EF_Cons_Registre_Soufflage
                Image (0,0 115x210), invisible if: NOT EF_Cons_Registre_Soufflage, image: ImagePool_Buttons.Red_Top
                    OnMouseDown: toggle EF_Cons_Registre_Soufflage
            Rectangle (115,0 132x57), "FORCE"
            Rectangle (112,76 132x57), "MODE"
            Rectangle (115,153 132x57), "NORMAL"
    Button (650,130 160x60), "Suivant"
        OnMouseDown: execute {
            IF (Option_Douche OR Option_Lavabo)
            	THEN
            	VisuElems.CURRENTVISU := 'Maintenance_2';
            	ELSIF (Option_Bas_Debit OR Option_Douchette OR Option_NEP)
            		THEN
            		VisuElems.CURRENTVISU := 'Maintenance_3';
            	ELSIF (Option_WC_GV OR Option_WC_PV OR Option_Prise)
            		THEN
            		VisuElems.CURRENTVISU := 'Maintenance_4';
            	ELSIF (Option_Cabine_Climatique)
            		THEN
            		VisuElems.CURRENTVISU := 'Maintenance_5';
            	ELSIF (Option_Com_RegSouf_Ultrason)
            		THEN
            		VisuElems.CURRENTVISU := 'Maintenance_6';
            	ELSE
            		VisuElems.CURRENTVISU := 'Maintenance_7';
            END_IF
        }
    Group (24,246 390x500)
        Rectangle (3,0 380x76), "Extraction"
        Group (72,64 246x208)
            Group (0,0 115x210)
                Image (0,0 115x210), invisible if: EF_Cons_Reg_Etanche_Ext, image: ImagePool_Buttons.Green_Bottom
                    OnMouseDown: toggle EF_Cons_Reg_Etanche_Ext
                Image (0,0 115x210), invisible if: NOT EF_Cons_Reg_Etanche_Ext, image: ImagePool_Buttons.Red_Top
                    OnMouseDown: toggle EF_Cons_Reg_Etanche_Ext
            Rectangle (115,0 132x57), "FORCE"
            Rectangle (112,76 132x57), "MODE"
            Rectangle (115,153 132x57), "NORMAL"
        Rectangle (0,349 390x76), "Appli : %.0f %%", text variable: Cons_Actionneur_Reg_Etanche_Ext
        Rectangle (0,424 390x76), "Mesure : %.0f %%", text variable: MES_Pos_Reg_Etanche_Ext
        RoundedRectangle (0,272 390x76), "Ouverture : %.0f %%", text variable: F_Cons_Reg_Etanche_Ext, invisible if: NOT EF_Cons_Reg_Etanche_Ext
            OnMouseDown: write the text variable via VisuDialogs.Numpad, min 0, max 100, format %.0f
    Group (868,246 390x500), invisible if: NOT Option_V3V_EauMitig
        Rectangle (3,0 380x76), "Vanne eau mitigée"
        Group (72,64 246x208)
            Group (0,0 115x210)
                Image (0,0 115x210), invisible if: EF_Cons_V3V_Eau_Mitig, image: ImagePool_Buttons.Green_Bottom
                    OnMouseDown: toggle EF_Cons_V3V_Eau_Mitig
                Image (0,0 115x210), invisible if: NOT EF_Cons_V3V_Eau_Mitig, image: ImagePool_Buttons.Red_Top
                    OnMouseDown: toggle EF_Cons_V3V_Eau_Mitig
            Rectangle (115,0 132x57), "FORCE"
            Rectangle (112,76 132x57), "MODE"
            Rectangle (115,153 132x57), "NORMAL"
        Rectangle (0,349 390x76), "Appli : %.0f %%", text variable: Cons_Actionneur_V3V_Eau_Mitig
        Rectangle (0,424 390x76), "Mesure : %.0f %%", text variable: Cons_Actionneur_V3V_Eau_Mitig, invisible if: TRUE
        RoundedRectangle (0,272 390x76), "Ouverture : %.0f %%", text variable: F_Cons_V3V_Eau_Mitig, invisible if: NOT EF_Cons_V3V_Eau_Mitig
            OnMouseDown: write the text variable via VisuDialogs.Numpad, min 0, max 100, format %.0f
END_VISUALIZATION

// ---- Visualizations/Visualizations/menu.TcVIS
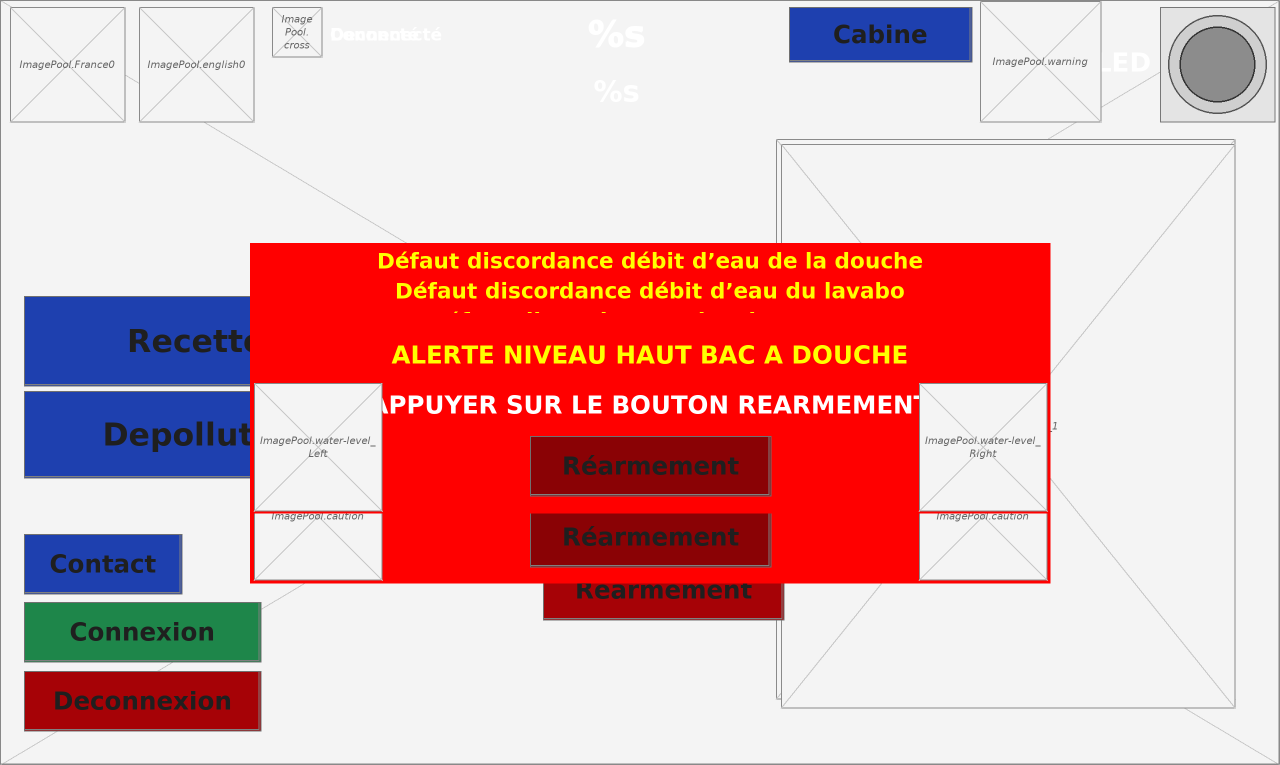
VISUALIZATION menu  // 1280x765
    Frame (0,0 1280x765)
        shows masque()
    Image (776,139 459x560), image: ImagePool.Cabine-2
    Polygon (802,613) (940,653) (1079,687) (1152,653) (1225,613), colour variable: GVL_Visu.Couleur_Cabine
    Polygon (804,613) (802,215) (1081,156) (1222,222) (1223,613), colour variable: GVL_Visu.Couleur_Cabine
    Button (24,391 363x87), "Depollution"
        OnMouseDown: change screen: Depollution
    Button (24,602 237x60), "Connexion"
        OnMouseDown: VisuUserMgmt Type=Login
    Button (24,296 363x90), "Recettes"
        OnMouseDown: change screen: Sel_Recettes
    Image (781,144 454x564), image: ImagePool.Cabine_1
        OnMouseDown: OpenDialog Dialog=Actionneurs, OpenModal=True, OpenCentered=True
    Group (387,389 372x89)
        Button (9,2 363x87), "Maintenance"
            OnMouseDown: execute {
                IF (Option_RegSouf_Ultrason OR Option_Reg_Etanche_Ext OR Option_V3V_EauMitig)
                	THEN
                	VisuElems.CURRENTVISU := 'Maintenance_1';
                	ELSIF (Option_Douche OR Option_Lavabo)
                		THEN
                		VisuElems.CURRENTVISU := 'Maintenance_2';
                	ELSIF (Option_Bas_Debit OR Option_Douchette OR Option_NEP)
                		THEN
                		VisuElems.CURRENTVISU := 'Maintenance_3';
                	ELSIF (Option_WC_GV OR Option_WC_PV OR Option_Prise)
                		THEN
                		VisuElems.CURRENTVISU := 'Maintenance_4';
                	ELSIF (Option_Cabine_Climatique)
                		THEN
                		VisuElems.CURRENTVISU := 'Maintenance_5';
                	ELSE
                	VisuElems.CURRENTVISU := 'Maintenance_6';
                END_IF
            }
        Image (0,0 79x74), invisible if: NOT GVL_Visu.Etat_Connexion, image: VisuSymbols.Symbols.LockOpen
        Image (8,0 79x74), invisible if: GVL_Visu.Etat_Connexion, image: VisuSymbols.Symbols.Lock
    Button (24,671 237x60), "Deconnexion"
        OnMouseDown: VisuUserMgmt Type=Logout
    Button (24,534 158x60), "Contact"
        OnMouseDown: change screen: Accueil
    Button (543,560 241x60), "Réarmement", invisible if: NOT Condi_Affich_Rearm
        OnMouseDown: toggle Cmd_Rearmement
    Group (816,245 317x202)
        Rectangle (6,162 290x40), "Eau : %.1f °C", text variable: MES_Temp_Eau_Mitige_General
        Rectangle (13,40 290x40), "Hygro : %.1f %Hr", text variable: Tab_MES_Sonde_Hygro_Amb.R_MesCor
        Rectangle (27,81 290x40), "Temp : %.1f °C", text variable: Tab_MES_Sonde_Temp_Amb.R_MesCor
        Rectangle (0,0 290x40), "Air : %.1f Vol/h", text variable: MES_Debit_Volh_Soufflage, invisible if: TRUE
        Rectangle (21,121 290x40), "Press : %.0f Pa", text variable: Tab_MES_Sonde_Press_Cab.R_MesCor
    Button (396,296 363x90), "Mode manuel"
        OnMouseDown: change screen: ModeManuel
    Group (250,243 800x340)
        Frame (0,0 800x340), invisible if: NOT GVL_Visu.Affichage_PopUp_Alarm
            shows PopUp_Alarms()
        Frame (0,70 800x200), invisible if: NOT GVL_Visu.Affichage_PopUp_HightLevel
            shows PopUp_Hight_Level()
END_VISUALIZATION

// ---- Visualizations/Visualizations/Mes_Textes/Etats_Cabine.TcTLO
TEXTLIST Etats_Cabine
  0 = 'CABINE EN DEFAUT' | En: 'FAULTY BOOTH'
  1 = 'CABINE LIBRE' | En: 'STANDBY'
  2 = 'MODE MANUEL EN COURS' | En: 'MANUAL MODE IN PROGRESS'
  3 = 'RECETTE EN COURS' | En: 'PROTOCOL IN PROGRESS'
  4 = 'MODE DEPOLLUTION EN COURS' | En: 'DECONTAMINATION IN PROGRESS'
  5 = 'MODE NETTOYAGE EN COURS' | En: 'CLEANING IN PROGRESS'
  6 = 'MODE ECO EN COURS' | En: 'ECO MODE IN PROGRESS'
  7 = 'MODE MAINTENANCE' | En: 'MAINTENANCE MODE'
  8 = 'MODE STOP' | En: 'STOP MODE'
   = ''
END_TEXTLIST

// ---- Visualizations/Visualizations/Objets/Door.TcVIS
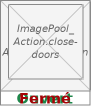
VISUALIZATION Door  // 91x106
VAR_IN_OUT
	Etat_MaAr	:BOOL;
END_VAR
    Rectangle (15,91 60x15), "Ouvert", invisible if: Etat_MaAr, text list: 'OuvFerm', text index: S_Cmd_ElectroValve_Alim_Lavabo
    Rectangle (15,91 60x15), "Fermé", invisible if: NOT Etat_MaAr, text list: 'OuvFerm', text index: S_Cmd_ElectroValve_Alim_Lavabo
    Image (0,0 91x91), invisible if: Etat_MaAr, image: ImagePool_Action.door-open
    Image (8,4 75x75), invisible if: NOT Etat_MaAr, image: ImagePool_Action.close-doors
END_VISUALIZATION

// ---- Visualizations/Visualizations/Objets/Sink.TcVIS
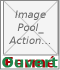
VISUALIZATION Sink  // 60x70
VAR_IN_OUT
	Etat_MaAr	:BOOL;
END_VAR
    Image (3,0 55x55), invisible if: NOT Etat_MaAr, image: ImagePool_Action.Sink_Open
    Image (3,0 55x55), invisible if: Etat_MaAr, image: ImagePool_Action.Sink_Close
    Rectangle (0,55 60x15), "Fermé", invisible if: Etat_MaAr, text list: 'OuvFerm', text index: S_Cmd_ElectroValve_Alim_Lavabo
    Rectangle (0,55 60x15), "Ouvert", invisible if: NOT Etat_MaAr, text list: 'OuvFerm', text index: S_Cmd_ElectroValve_Alim_Lavabo
END_VISUALIZATION

// ---- Visualizations/Visualizations/Objets/Drain.TcVIS
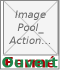
VISUALIZATION Drain  // 60x70
VAR_IN_OUT
	Etat_MaAr	:BOOL;
END_VAR
    Rectangle (0,55 60x15), "Fermé", invisible if: Etat_MaAr, text list: 'OuvFerm', text index: S_Cmd_ElectroValve_Alim_Lavabo
    Rectangle (0,55 60x15), "Ouvert", invisible if: NOT Etat_MaAr, text list: 'OuvFerm', text index: S_Cmd_ElectroValve_Alim_Lavabo
    Image (3,0 55x55), invisible if: Etat_MaAr, image: ImagePool_Action.drain_Close
    Image (3,0 55x55), invisible if: NOT Etat_MaAr, image: ImagePool_Action.drain_Open
END_VISUALIZATION

// ---- Visualizations/Visualizations/Objets/Plug.TcVIS
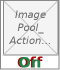
VISUALIZATION Plug  // 60x70
VAR_IN_OUT
	Etat_MaAr	:BOOL;
END_VAR
    Rectangle (0,55 60x15), "Off", invisible if: Etat_MaAr, text list: 'OuvFerm', text index: S_Cmd_ElectroValve_Alim_Lavabo
    Rectangle (0,55 60x15), "On", invisible if: NOT Etat_MaAr, text list: 'OuvFerm', text index: S_Cmd_ElectroValve_Alim_Lavabo
    Image (3,0 55x55), invisible if: Etat_MaAr, image: ImagePool_Action.Plug_Offe
    Image (3,0 55x55), invisible if: NOT Etat_MaAr, image: ImagePool_Action.Plug_On
END_VISUALIZATION

// ---- Visualizations/Visualizations/PopUp/Actionneurs.TcVIS
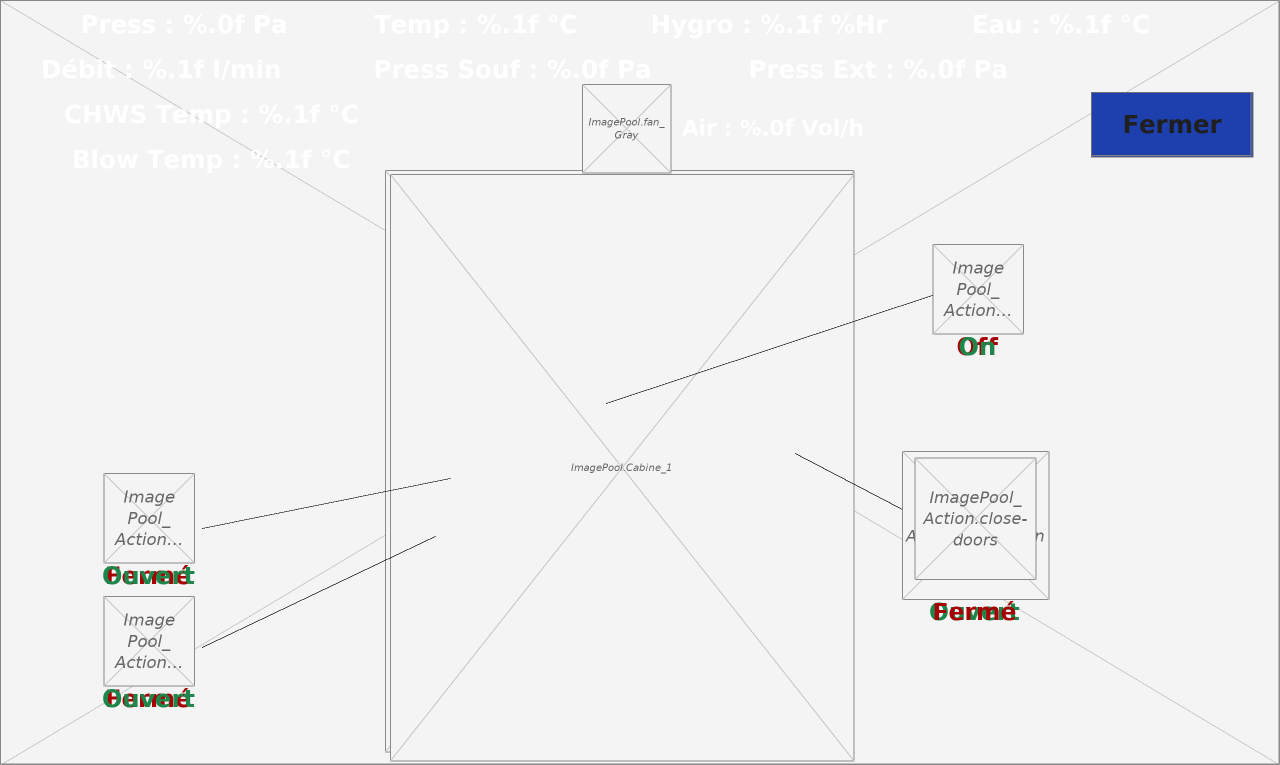
VISUALIZATION Actionneurs  // 1280x765
    Image (0,0 1280x765), image: ImagePool.Fond_Degr
    Image (385,170 469x582), image: ImagePool.Cabine-2
    Polygon (412,662) (553,704) (695,739) (769,704) (844,662), colour variable: GVL_Visu.Couleur_Cabine
    Polygon (414,662) (412,248) (697,187) (840,256) (842,662), colour variable: GVL_Visu.Couleur_Cabine
    Image (390,174 464x587), image: ImagePool.Cabine_1
    Line (202,528) (450,478)
    Line (795,453) (929,523)
    Line (606,403) (941,292)
    Button (1091,92 162x65), "Fermer"
        OnMouseDown: CloseDialog Dialog=Actionneurs, Result=OK, NumpadKeypadSet=True
    Group (582,84 393x89), invisible if: TRUE
        Rectangle (97,23 296x42), "Air : %.0f Vol/h", text variable: MES_Debit_Volh_Soufflage
        Group (0,0 89x89), invisible if: NOT Visu.On_Off_Ventilation
            Image (0,0 55x55), invisible if: NOT GVL_Visu.On_Off_Anim, image: ImagePool.fan_45
            Image (0,0 55x55), invisible if: GVL_Visu.On_Off_Anim, image: ImagePool.fan (1)
        Image (0,0 89x89), invisible if: Visu.On_Off_Ventilation, image: ImagePool.fan_Gray
    Frame (99,473 99x115)
        shows Sink(Etat_MaAr := S_Cmd_ElectroValve_Alim_Lavabo)
    Line (202,647) (435,536)
    Frame (902,451 147x173)
        shows Door(Etat_MaAr := E_Info_Contact_Porte)
    Frame (928,244 99x115)
        shows Plug(Etat_MaAr := S_Cmd_PC_Cab)
    Frame (99,596 99x115)
        shows Drain(Etat_MaAr := S_Cmd_Vanne_Vid_Lavabo)
    Rectangle (623,2 292x45), "Hygro : %.1f %Hr", text variable: Tab_MES_Sonde_Hygro_Amb.R_MesCor
    Rectangle (330,2 292x45), "Temp : %.1f °C", text variable: Tab_MES_Sonde_Temp_Amb.R_MesCor
    Rectangle (38,2 292x45), "Press : %.0f Pa", text variable: Tab_MES_Sonde_Press_Cab.R_MesCor
    Rectangle (915,2 292x45), "Eau : %.1f °C", text variable: MES_Temp_Eau_Mitige_General
    Rectangle (38,47 292x45), "Débit : %.1f l/min", text variable: GVL_Visu.Visu_Mes_Debit_Eau_Manu, invisible if: NOT a5_Ecriture_InterCom.Dmd_Mise_En_Temp
    Rectangle (330,47 365x45), "Press Souf : %.0f Pa", text variable: Tab_Mes_Sonde_Pression_Souf.R_MesCor, invisible if: NOT Option_Press_SoufExt_General
    Rectangle (696,47 365x45), "Press Ext : %.0f Pa", text variable: Tab_Mes_Sonde_Pression_Ext.R_MesCor, invisible if: NOT Option_Press_SoufExt_General
    Rectangle (38,92 347x45), "CHWS Temp : %.1f °C", text variable: Tab_Mes_Sonde_Temp_BatEG.R_MesCor
    Rectangle (38,137 347x45), "Blow Temp : %.1f °C", text variable: Tab_Mes_Sonde_Temp_Souf.R_MesCor
END_VISUALIZATION

// ---- Visualizations/Visualizations/PopUp/Alarmes.TcVIS
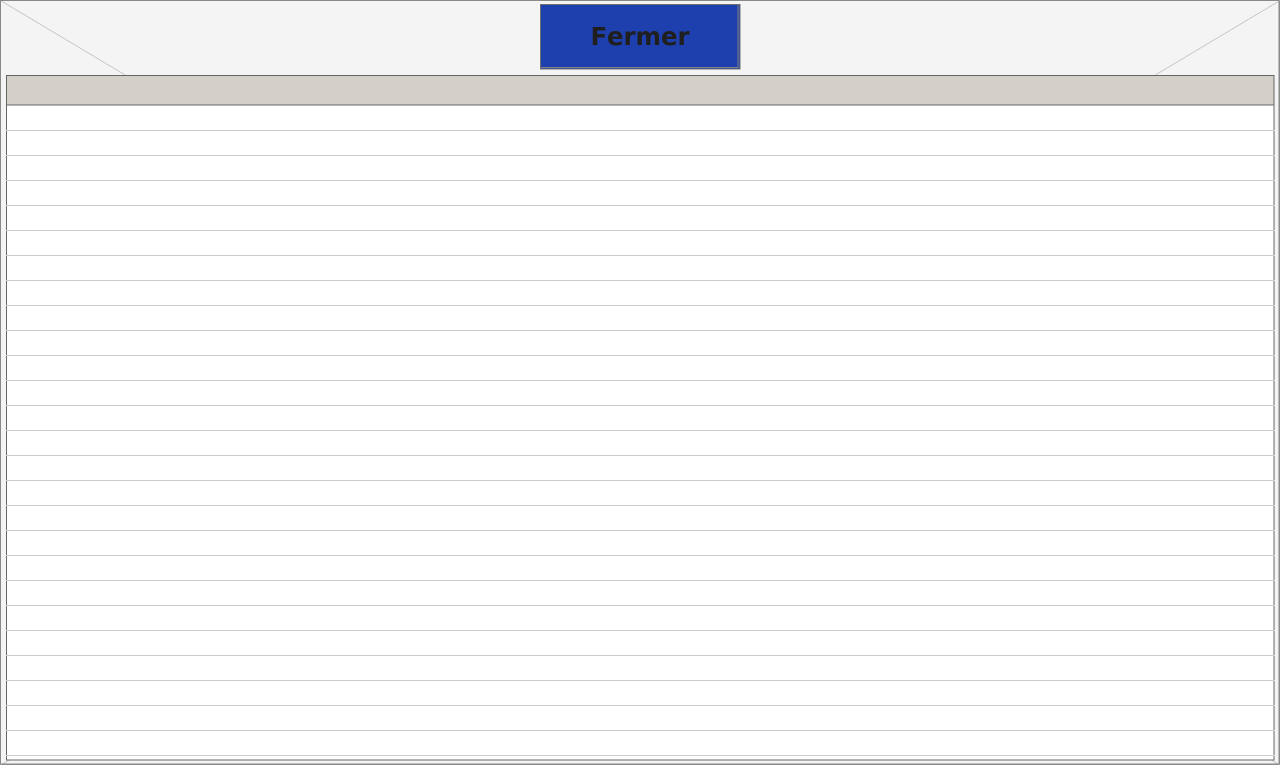
VISUALIZATION Alarmes  // 1280x765
    Image (0,0 1280x765), image: ImagePool.Fond_Degr
    Button (540,4 200x65), "Fermer"
        OnMouseDown: CloseDialog Dialog=Alarmes, Result=OK, NumpadKeypadSet=True
    Table (6,75 1268x685), invisible if: VisuElems.CURRENTLANGUAGE = 'en', data array: Alarmes.Tab_Alarme_FREN
        p3854506369: Alarmes.Tab_Alarme_FREN[1,INDEX]
        p1892666644: Alarmes.Tab_Alarme_FREN[2,INDEX]
    Table (6,75 1268x685), invisible if: VisuElems.CURRENTLANGUAGE = 'fr', data array: Alarmes.Tab_Alarme_FREN
        p3854506369: Alarmes.Tab_Alarme_FREN[1,INDEX]
        p1892666644: Alarmes.Tab_Alarme_FREN[2,INDEX]
END_VISUALIZATION

// ---- Visualizations/Visualizations/PopUp/PopUp_Alarms.TcVIS
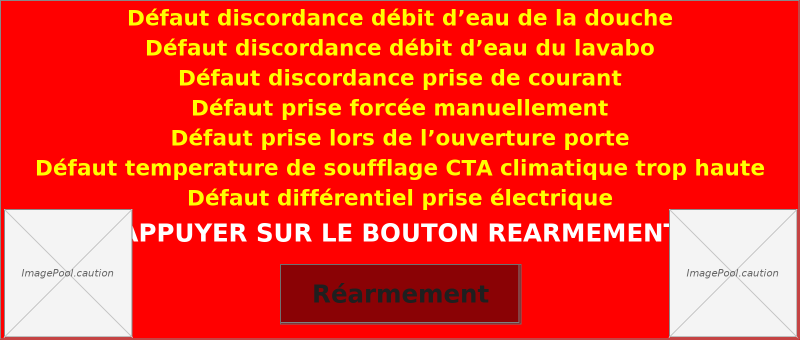
VISUALIZATION PopUp_Alarms  // 800x340
    RoundedRectangle (0,3 800x30), "Défaut discordance débit d’eau de la douche", invisible if: NOT Defaut_Discord_Deb_Eau_Douche
    Button (280,264 241x60), "Réarmement", invisible if: NOT Condi_Affich_Rearm
        OnMouseDown: toggle Cmd_Rearmement
    RoundedRectangle (0,208 800x50), "APPUYER SUR LE BOUTON REARMEMENT"
    Image (4,209 128x128), image: ImagePool.caution
    Image (669,209 128x128), image: ImagePool.caution
    RoundedRectangle (0,33 800x30), "Défaut discordance débit d’eau du lavabo", invisible if: NOT Defaut_Discord_Deb_Eau_Lavabo
    RoundedRectangle (0,63 800x30), "Défaut discordance prise de courant", invisible if: NOT Defaut_Discord_PC_Cab
    RoundedRectangle (0,93 800x30), "Défaut prise forcée manuellement", invisible if: NOT Def_Discord_Alim_Prise
    RoundedRectangle (0,123 800x30), "Défaut prise lors de l’ouverture porte", invisible if: NOT Def_Prise_Porte_Ouverte
    RoundedRectangle (0,183 800x30), "Défaut différentiel prise électrique", invisible if: NOT Defaut_Differentiel_Prise_Elec
    RoundedRectangle (0,153 800x30), "Défaut temperature de soufflage CTA climatique trop haute", invisible if: NOT Defaut_Thermostat_Secu
END_VISUALIZATION

// ---- Visualizations/Visualizations/PopUp/PopUp_Hight_Level.TcVIS
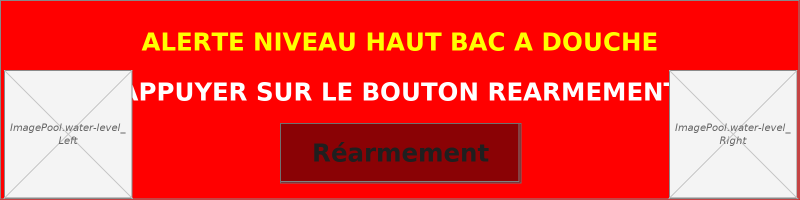
VISUALIZATION PopUp_Hight_Level  // 800x200
    Button (280,123 241x60), "Réarmement", invisible if: NOT Condi_Affich_Rearm
        OnMouseDown: toggle Cmd_Rearmement
    RoundedRectangle (0,17 800x50), "ALERTE NIVEAU HAUT BAC A DOUCHE"
    RoundedRectangle (0,67 800x50), "APPUYER SUR LE BOUTON REARMEMENT"
    Image (4,70 128x128), image: ImagePool.water-level_Left
    Image (669,70 128x128), image: ImagePool.water-level_Right
END_VISUALIZATION

// ---- Visualizations/Visualizations/Recet_EnCours.TcVIS
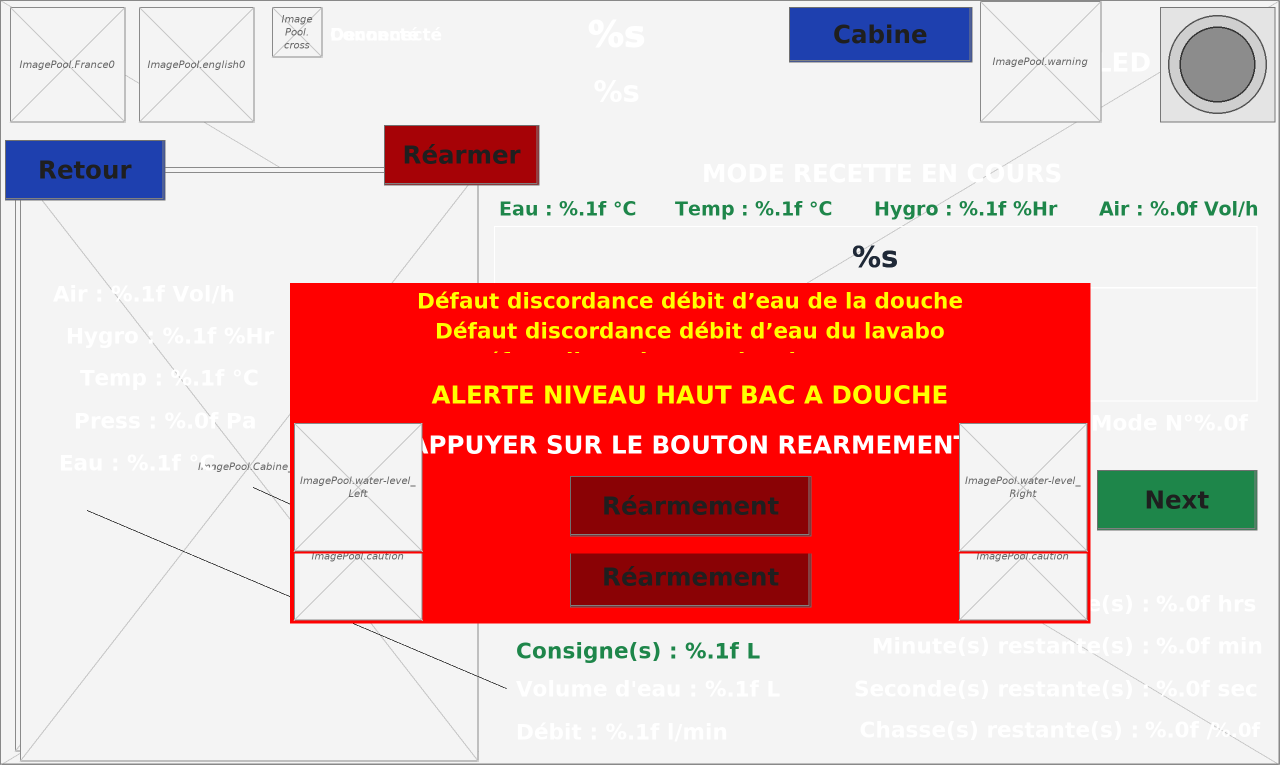
VISUALIZATION Recet_EnCours  // 1280x765
    Frame (0,0 1280x765)
        shows masque()
    Group (494,149 763x386), invisible if: NOT Mode_Cabine_Automatique
        Button (0,321 160x60), "Stop"
            OnMouseDown: toggle Reset_Mode_Auto
        Rectangle (81,0 615x49), "MODE RECETTE EN COURS", invisible if: GVL_Visu.On_Off_Anim
        Button (603,321 160x60), "Next", invisible if: NOT Condi_Affich_Etape_Suiv
            OnMouseDown: toggle Valid_Texte
        Button (302,321 160x60), "Re-Start", invisible if: NOT Statut_Pause_Force
            OnMouseDown: toggle Bp_Pause
    Image (15,167 463x584), image: ImagePool.Cabine-2
    Polygon (42,662) (181,704) (321,739) (395,704) (468,662), colour variable: GVL_Visu.Couleur_Cabine
    Polygon (44,662) (42,246) (323,185) (465,254) (467,662), colour variable: GVL_Visu.Couleur_Cabine
    Image (20,172 458x589), image: ImagePool.Cabine_1
        OnMouseDown: OpenDialog Dialog=Actionneurs, OpenModal=True, OpenCentered=True
    Group (834,583 431x127), invisible if: NOT GVL_Visu.Visu_Tempo
        Rectangle (0,0 319x42), "Heure(s) restante(s) :"
        Rectangle (319,0 112x42), "%.0f hrs", text variable: Temp_Restant_Heure
        Rectangle (0,85 319x42), "Seconde(s) restante(s) :"
        Rectangle (319,85 112x42), "%.0f sec", text variable: Temp_Restant_Seconde
        Rectangle (0,42 319x42), "Minute(s) restante(s) :"
        Rectangle (319,42 112x42), "%.0f min", text variable: Temp_Restant_Minute
    Button (5,140 160x60), "Retour", invisible if: Mode_Cabine_Automatique
        OnMouseDown: change screen: menu
    Rectangle (496,402 176x42), "Etape : %d /", text variable: Numero_Etape_Actuel
    Rectangle (676,402 112x42), "%d", text variable: Nbre_Etape_Totale
    Rectangle (1075,402 176x42), "Mode N°%.0f", text variable: Numero_Mode_Actuel
    Group (494,226 763x62)
        RoundedRectangle (0,0 763x62)
        Rectangle (0,0 763x62), "%s", text variable: Tab_Nom_Recette[1,0], invisible if: VisuElems.CURRENTLANGUAGE = 'en'
        Rectangle (0,0 763x62), "%s", text variable: Tab_Nom_Recette[2,0], invisible if: VisuElems.CURRENTLANGUAGE = 'fr'
    Group (494,287 763x114)
        RoundedRectangle (0,0 763x114)
        Rectangle (0,0 763x114), "%s", text variable: Lecture_Texte_Choisi_FR, invisible if: VisuElems.CURRENTLANGUAGE = 'en'
        Rectangle (0,0 763x114), "%s", text variable: Lecture_Texte_Choisi_ENG, invisible if: VisuElems.CURRENTLANGUAGE = 'fr'
    Group (496,192 777x34)
        Rectangle (0,0 171x34), "Eau : %.1f °C", text variable: n3_Regul_Temp_EauMitig.SetPoint_PID_Temp_EM, invisible if: NOT a5_Ecriture_InterCom.Dmd_Mise_En_Temp
        Rectangle (176,0 196x34), "Temp : %.1f °C", text variable: Lect_Cons_Temperature_Cabine, invisible if: NOT RS_MEnCond.Q1
        Rectangle (375,0 233x34), "Hygro : %.1f %Hr", text variable: Lect_Cons_Hygrometrie_Cabine, invisible if: NOT RS_MEnCond.Q1
        Rectangle (600,0 177x34), "Air : %.0f Vol/h", text variable: Cons_Actionneur_Registre_Souf_Volh
    Group (823,709 442x42), invisible if: NOT GVL_Visu.Visu_ChasseEau
        Rectangle (0,0 319x42), "Chasse(s) restante(s) :"
        Rectangle (319,0 73x42), "%.0f /", text variable: Nbre_Chasse_EnCours
        Rectangle (385,0 57x42), "%.0f", text variable: Nbre_Chasse_Total
    Group (253,487 602x140), invisible if: NOT GVL_Visu.Visu_VolEau_Douche
        Line (0,0) (255,115)
        Rectangle (260,98 342x42), "Volume d'eau : %.1f L", text variable: Lect_Volume_Eau_Douche
        Rectangle (260,63 342x34), "Consigne(s) : %.1f L", text variable: Cons_Volume_Eau_Douche_Actuel
    Group (87,510 768x200), invisible if: NOT GVL_Visu.Visu_VolEau_Lavabo
        Line (0,0) (419,178)
        Rectangle (426,158 342x42), "Volume d'eau : %.1f L", text variable: Lect_Volume_Eau_Lavabo
        Rectangle (426,124 342x34), "Consigne(s) : %.1f L", text variable: Cons_Volume_Eau_Lavabo_Actuel
    Button (384,125 155x60), "Réarmer", invisible if: NOT Condi_Affich_Rearm
        OnMouseDown: toggle Cmd_Rearmement
    Group (50,273 319x211)
        Rectangle (13,42 292x42), "Hygro : %.1f %Hr", text variable: Tab_MES_Sonde_Hygro_Amb.R_MesCor
        Rectangle (27,84 292x42), "Temp : %.1f °C", text variable: Tab_MES_Sonde_Temp_Amb.R_MesCor
        Rectangle (0,0 292x42), "Air : %.1f Vol/h", text variable: MES_Debit_Volh_Soufflage, invisible if: TRUE
        Rectangle (21,127 292x42), "Press : %.0f Pa", text variable: Tab_MES_Sonde_Press_Cab.R_MesCor
        Rectangle (6,169 292x42), "Eau : %.1f °C", text variable: MES_Temp_Eau_Mitige_General
    Rectangle (513,711 292x42), "Débit : %.1f l/min", text variable: GVL_Visu.Visu_Mes_Debit_Eau, invisible if: NOT GVL_Visu.Visu_Debit_Eau
    Group (290,283 800x340)
        Frame (0,0 800x340), invisible if: NOT GVL_Visu.Affichage_PopUp_Alarm
            shows PopUp_Alarms()
        Frame (0,70 800x200), invisible if: NOT GVL_Visu.Affichage_PopUp_HightLevel
            shows PopUp_Hight_Level()
END_VISUALIZATION

// ---- Visualizations/Visualizations/Sel_Recettes.TcVIS
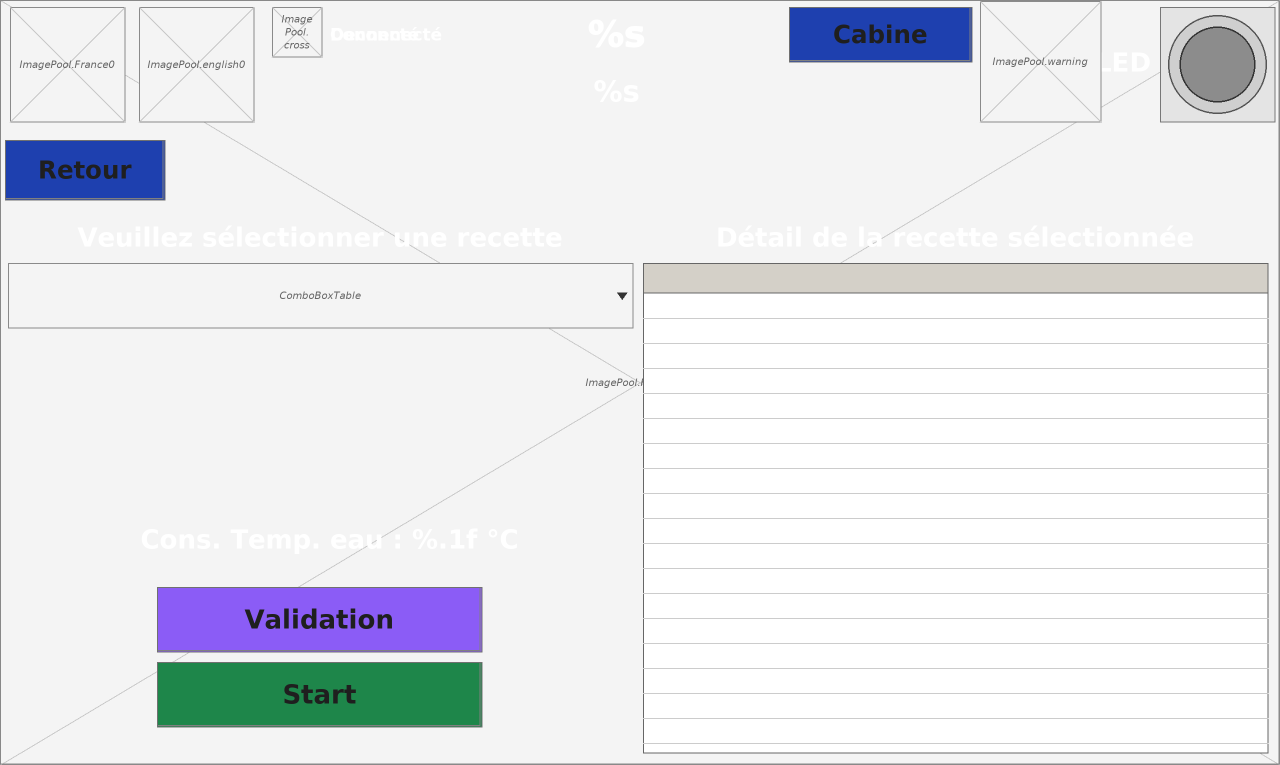
VISUALIZATION Sel_Recettes  // 1280x765
    Frame (0,0 1280x765)
        shows masque()
    ComboBoxTable (8,263 625x65), variable: Numero_Recette_Sel, invisible if: VisuElems.CURRENTLANGUAGE = 'en', data array: Tab_Nom_Recette
        p3854506369: Tab_Nom_Recette[1,INDEX]
        p1892666644: Tab_Nom_Recette[2,INDEX]
    Button (5,140 160x60), "Retour"
        OnMouseDown: change screen: menu
    ComboBoxTable (8,263 625x65), variable: Numero_Recette_Sel, invisible if: VisuElems.CURRENTLANGUAGE = 'fr', data array: Tab_Nom_Recette
        p3854506369: Tab_Nom_Recette[1,INDEX]
        p1892666644: Tab_Nom_Recette[2,INDEX]
    Table (643,263 625x490), invisible if: VisuElems.CURRENTLANGUAGE = 'en', data array: Tab_Nom_Mode
        p3854506369: Tab_Nom_Mode[1,INDEX]
        p1892666644: Tab_Nom_Mode[2,INDEX]
    Rectangle (39,213 562x49), "Veuillez sélectionner une recette", text variable: MES_Debit_Volh_Soufflage
    Rectangle (674,213 562x49), "Détail de la recette sélectionnée", text variable: MES_Debit_Volh_Soufflage
    Table (643,263 625x490), invisible if: VisuElems.CURRENTLANGUAGE = 'fr', data array: Tab_Nom_Mode
        p3854506369: Tab_Nom_Mode[1,INDEX]
        p1892666644: Tab_Nom_Mode[2,INDEX]
    Button (157,587 325x65), "Validation"
        OnMouseDown: toggle Validation_Recette_Auto
    Button (157,662 325x65), "Start", invisible if: GVL_Visu.Visu_Btn_Start
        OnMouseDown: change screen: Recet_EnCours
        OnMouseDown: toggle Start_Recette_Mode_Auto
    RoundedRectangle (118,507 423x65), "Cons. Temp. eau : %.1f °C", text variable: Cons_Temp_EauMitige, invisible if: NOT Option_Regul_Temp_Eau
        OnMouseDown: write the text variable via VisuDialogs.Numpad, min 0, max 50, format %.0f
END_VISUALIZATION
